(* PLC project factoryx.project, Bedrock IDE Bedrock IDE V1.4 *)
(* stored: creationDateTime 2017-02-21T09:02:52.9855728, modificationDateTime 2017-02-21T09:02:15.4674269 *)

TYPE EM_I_OUT_COM : STRUCT
  Request : INT;
  Command : INT;
  Pressure_SP : REAL;
  Owner : INT;
  Status : INT;
  CM_error : BOOL;
  CM_error_no : DINT;
  q_bACTVIE : BOOL;
  Level : REAL;
  Pressure : REAL;
END_STRUCT;
END_TYPE

FUNCTION somefunction : INT
  VAR_INPUT
    arg1 : INT;
    arg2 : INT;
  END_VAR

            
          
END_FUNCTION

FUNCTION write_to_DB_DW : BOOL
  VAR_INPUT
    DB_NO : INT;
    Location : INT;
    Value : INT;
  END_VAR

            
          
END_FUNCTION

FUNCTION_BLOCK Valve
  VAR_INPUT
    Command : BOOL;
    Feedback_Open : BOOL;
    Feedback_Close : BOOL;
  END_VAR
  VAR_OUTPUT
    Opened : BOOL;
    Closed : BOOL;
    Monitoring_Error : BOOL;
    Command_Open : BOOL;
  END_VAR

                    
                  
END_FUNCTION_BLOCK

FUNCTION_BLOCK Motor
  VAR_INPUT
    Command_On : BOOL;
    Command_Off : BOOL;
    Auto : BOOL;
    Manual : BOOL;
    Feedback_On : BOOL;
    Remote : BOOL;
    Error : BOOL;
    Enable : BOOL;
    Repair : BOOL;
  END_VAR
  VAR_OUTPUT
    Running : BOOL;
    Stopped : BOOL;
    Command_Run : BOOL;
    Error_Mon : BOOL;
    Error_VFD : BOOL;
    Error_Out : BOOL;
  END_VAR

                    
                  
END_FUNCTION_BLOCK

FUNCTION_BLOCK Motor_VFD
  VAR_INPUT
    Command_On : BOOL;
    Command_Off : BOOL;
    Auto : BOOL;
    Manual : BOOL;
    Feedback_On : BOOL;
    Remote : BOOL;
    Error : BOOL;
    Enable : BOOL;
    Repair : BOOL;
  END_VAR
  VAR_OUTPUT
    Running : BOOL;
    Stopped : BOOL;
    Command_Run : BOOL;
    Error_MS : BOOL;
    Error_Out : BOOL;
  END_VAR

                    
                  
END_FUNCTION_BLOCK

FUNCTION_BLOCK AI
  VAR_INPUT
    wVal : REAL;
  END_VAR
  VAR_OUTPUT
    QfVal : REAL;
    LIM_QbAH : BOOL;
    LIM_QbWH : BOOL;
    LIM_QbWL : BOOL;
    LIM_QbAL : BOOL;
    QERR : BOOL;
  END_VAR

                    
                  
END_FUNCTION_BLOCK

FUNCTION_BLOCK DI
  VAR_INPUT
    i_bInp : BOOL;
  END_VAR
  VAR_OUTPUT
    QON : BOOL;
  END_VAR

                    
                  
END_FUNCTION_BLOCK

FUNCTION_BLOCK PID
  VAR_INPUT
    i_bPCmdAUT : BOOL;
    i_bPCmdMAN : BOOL;
    Operator_Setpoint : REAL;
    Set_SP : BOOL;
    i_bPCmdPID : BOOL;
    i_bPCmdOPE : BOOL;
    Output_Value : REAL;
    Set_Output : REAL;
    wVal : REAL;
  END_VAR
  VAR_OUTPUT
    QfVal : REAL;
    QERR : BOOL;
    Q_wOP : REAL;
  END_VAR

                    
                  
END_FUNCTION_BLOCK

FUNCTION_BLOCK EM_I_OUT
  VAR_INPUT
    scantime : REAL := 200.0;
    sampletime : REAL;
    em_id : INT;
    Request : INT;
    Command : INT;
    Pressure_SP : REAL;
    Pump_RUN : BOOL;
    Pump_QERR : BOOL;  (* - General Error *)
    Pump_EERR : BOOL;  (* - External Error *)
    FS01_PV : BOOL;  (* Flow Switch - Digital Measurement *)
    PIC01_PV : REAL;  (* Pressure Controller *)
    PIC01_ERR : BOOL;  (* Pressure Controller *)
    LT01_PV : REAL;  (* Level Transmitter (m) *)
    LT01_AHH : BOOL;  (* Level Transmitter (m) *)
    LT01_AH : BOOL;  (* Level Transmitter (m) *)
    LT01_AL : BOOL;  (* Level Transmitter (m) *)
    LT01_ALL : BOOL;  (* Level Transmitter (m) *)
    LT01_ERR : BOOL;  (* Level Transmitter (m) *)
    XV_Bottom_OPN : BOOL;  (* Automatic Bottom Valve *)
    XV_Bottom_CLS : BOOL;  (* Automatic Bottom Valve *)
    XV_Bottom_MERR : BOOL;  (* Automatic Bottom Valve *)
    BV_Bottom_OPN : BOOL;  (* Manual Bottom Valve *)
    BV_Bottom_CLS : BOOL;  (* Manual Bottom Valve *)
    BV_Bottom_MERR : BOOL;  (* Manual Bottom Valve *)
    BV_Tran_M04_OPN : BOOL;  (* Trnasfer Valve to M04 *)
    BV_Tran_M04_CLS : BOOL;  (* Trnasfer Valve to M04 *)
    BV_Tran_M04_MERR : BOOL;  (* Trnasfer Valve to M04 *)
  END_VAR
  VAR_OUTPUT
    steptime_s : REAL;
    steptime_m : REAL;
    steptime_h : REAL;
    steptime_s : REAL;
    steptime_m : REAL;
    steptime_h : REAL;
    first_scan : BOOL;
    last_scan : BOOL;
    error_index_db : BOOL;
    Owner : INT;
    Status : INT;
    CM_error : BOOL;
    CM_error_no : DINT;
    q_bACTVIE : BOOL;
    Level : REAL;
    Pressure : REAL;
    Pump_ON : BOOL;  (* - Switch Motor ON *)
    Pump_AUT : BOOL;  (* - Swtich Motor to AUTO *)
    PIC01_EXT : BOOL;  (* Pressure Controller - Switch to External Mode *)
    PIC01_SP : REAL;  (* Pressure Controller - Operator Setpoint in Internal Mode *)
    PIC01_AUT : BOOL;  (* Pressure Controller - Switch to Auto Mode *)
    PIC01_VAL_OUT : REAL;  (* Pressure Controller - Operator Output Value *)
    PIC01_SET_SP : BOOL;  (* Pressure Controller *)
    PIC01_SET_OUT : BOOL;  (* Pressure Controller *)
    XV_Bottom_CMD : BOOL;  (* Automatic Bottom Valve - Auto command from program *)
    BV_Bottom_CMD : BOOL;  (* Manual Bottom Valve - Auto command from program *)
    BV_Tran_M04_CMD : BOOL;  (* Trnasfer Valve to M04 - Auto command from program *)
  END_VAR
  VAR
    first_scan : BOOL;
    last_scan : BOOL;
    previous_Command : INT;
    SP_PV : EM_I_OUT_COM;
  END_VAR
  VAR_TEMP
    initial_scan : BOOL;
  END_VAR

                    

					
// Copy all Setpoints from the COM
//--------------------------------
// 
//--------------------------------


Request:= SP_PV.Request;
Command:= SP_PV.Command;
Pressure_SP:= SP_PV.Pressure_SP;


// Acquiring logic
//--------------------------------
// 
//--------------------------------

Owner:= Request;


// Steptimers
//--------------------------------
// If the previous Command is not the same as the current one
// then reset the timers, else increase them
// This is at the start of the FB because normal commandchanges will take
// till the next cycle to become active
//--------------------------------

// if Command not changed then increase steptimer
IF (Command = previous_Command) THEN
	
	steptime_s:= steptime_s + scantime;

// else reset it at the start of a new step	
ELSE

	steptime_s:= 0.0;	
	
END_IF

// calculate the other two timers
steptime_m:= steptime_s / 60.0;
steptime_h:= steptime_m / 60.0;
		

		
// detect initial scan
//--------------------------------
// create a pulse active on the first cycle of a new scan
// this signal can be used in the step to execute some actions in the first cycle of the step
//--------------------------------

initial_scan:= Command <> previous_Command;		


// Save old step
//--------------------------------
// Save old step
//--------------------------------

previous_Command := Command;
		
		
// Collect the errors from the CMs
//--------------------------------
//
//--------------------------------
CM_Error:= (
	Pump_QERR
	OR Pump_EERR
	OR PIC01_ERR
	OR LT01_ERR
	OR XV_Bottom_MERR
	OR BV_Bottom_MERR
	OR BV_Tran_M04_MERR
);		
	

// Assign a message number to each error
//--------------------------------
// This code tries to assign an error message to each CM error
// If multiple CMs have an error then it only stores one
// This is the EM type so we don't know which CM/EM instance is connected
// So the error only contains the general name of the CM/EM instance
// If the actual name needs to be shown then it could be deducted
// at a higher level using the CM/EM name and EM instance 
//--------------------------------

// todo	


// START OF THE STATES
//################################
//################################
// Placeholder network to indicate the start of the actual sequence
//################################	  
//################################
// Step 0
//___EM_I_OUT_Step_0_
//================================
 
//================================	  

IF (Command = 0) THEN

	
	IF (first_scan) THEN
	
		// --- FIRST SCAN ---
		

	ELSE
	
		// --- CONTINUOUS ---
		

		// Action: stop Pump
		Pump_ON:= false;

		// Action: close XV_Bottom
		XV_Bottom_CMD:= false;

		// Action: close BV_Bottom
		BV_Bottom_CMD:= false;

		// Action: close BV_Tran_M04
		BV_Tran_M04_CMD:= false;

	END_IF
	

	// --- CONDITIONS ---
	IF (
		XV_Bottom_CLS
		AND BV_Bottom_CLS
		AND BV_Tran_M04_CLS
	) THEN
	
		Status:= Command;
		
	END_IF
	
END_IF	

IF (previous_Command = 0 and Command <> 0 ) THEN		
	
	
	// --- LAST SCAN ---
	


END_IF 

	
// Step 1
//___EM_I_OUT_Step_1_
//================================
 
//================================	  

IF (Command = 1) THEN

	
	IF (first_scan) THEN
	
		// --- FIRST SCAN ---
		

	ELSE
	
		// --- CONTINUOUS ---
		

		// Action: stop Pump
		Pump_ON:= false;

		// Action: open XV_Bottom
		XV_Bottom_CMD:= true;

	END_IF
	

	// --- CONDITIONS ---
	IF (
		XV_Bottom_OPN
	) THEN
	
		Status:= Command;
		
	END_IF
	
END_IF	

IF (previous_Command = 1 and Command <> 1 ) THEN		
	
	
	// --- LAST SCAN ---
	


END_IF 

	
// Step 2
//___EM_I_OUT_Step_2_
//================================
 
//================================	  

IF (Command = 2) THEN

	
	IF (first_scan) THEN
	
		// --- FIRST SCAN ---
		

		// Action: PIC01_SP = 10.0
		PIC01_SP:= 10.0;

		// Action: PIC01_SET_SP = true
		PIC01_SET_SP:= true;

	ELSE
	
		// --- CONTINUOUS ---
		

		// Action: start Pump
		Pump_ON:= true;

		// Action: auto 10.0 bar PIC01
		PIC01_AUT:= true;

		// Action: open XV_Bottom
		XV_Bottom_CMD:= true;

		// Action: PIC01_SET_SP = false
		PIC01_SET_SP:= false;

	END_IF
	

	// --- CONDITIONS ---
	IF (
		Pump_RUN
		AND XV_Bottom_OPN
	) THEN
	
		Status:= Command;
		
	END_IF
	
END_IF	

IF (previous_Command = 2 and Command <> 2 ) THEN		
	
	
	// --- LAST SCAN ---
	


END_IF 

	
// Step 3
//___EM_I_OUT_Step_3_
//================================
 
//================================	  

IF (Command = 3) THEN

	
	IF (first_scan) THEN
	
		// --- FIRST SCAN ---
		

	ELSE
	
		// --- CONTINUOUS ---
		

		// Action: stop Pump
		Pump_ON:= false;

		// Action: open BV_Bottom
		BV_Bottom_CMD:= true;

		// Action: open BV_Tran_M04
		BV_Tran_M04_CMD:= true;

	END_IF
	

	// --- CONDITIONS ---
	IF (
		BV_Bottom_OPN
		AND BV_Tran_M04_OPN
	) THEN
	
		Status:= Command;
		
	END_IF
	
END_IF	

IF (previous_Command = 3 and Command <> 3 ) THEN		
	
	
	// --- LAST SCAN ---
	


END_IF 

	
// Step 4
//___EM_I_OUT_Step_4_
//================================
 
//================================	  

IF (Command = 4) THEN

	
	IF (first_scan) THEN
	
		// --- FIRST SCAN ---
		

		// Action: PIC01_SP = Pressure_SP
		PIC01_SP:= Pressure_SP;

		// Action: PIC01_SET_SP = true
		PIC01_SET_SP:= true;

	ELSE
	
		// --- CONTINUOUS ---
		

		// Action: start Pump
		Pump_ON:= true;

		// Action: auto Pressure_SP PIC01
		PIC01_AUT:= true;

		// Action: open BV_Bottom
		BV_Bottom_CMD:= true;

		// Action: open BV_Tran_M04
		BV_Tran_M04_CMD:= true;

		// Action: PIC01_SET_SP = false
		PIC01_SET_SP:= false;

	END_IF
	

	// --- CONDITIONS ---
	IF (
		Pump_RUN
		AND BV_Bottom_OPN
		AND BV_Tran_M04_OPN
	) THEN
	
		Status:= Command;
		
	END_IF
	
END_IF	

IF (previous_Command = 4 and Command <> 4 ) THEN		
	
	
	// --- LAST SCAN ---
	


END_IF 

	
// Step 5
//___EM_I_OUT_Step_5_
//================================
 
//================================	  

IF (Command = 5) THEN

	
	IF (first_scan) THEN
	
		// --- FIRST SCAN ---
		

		// Action: PIC01_VAL_OUT = 20.0
		PIC01_VAL_OUT:= 20.0;

		// Action: PIC01_SET_OUT = true
		PIC01_SET_OUT:= true;

	ELSE
	
		// --- CONTINUOUS ---
		

		// Action: start Pump
		Pump_ON:= true;

		// Action: manual 20.0 Hz PIC01
		PIC01_AUT:= false;

		// Action: open XV_Bottom
		XV_Bottom_CMD:= true;

		// Action: PIC01_SET_OUT = false
		PIC01_SET_OUT:= false;

	END_IF
	

	// --- CONDITIONS ---
	IF (
		Pump_RUN
		AND XV_Bottom_OPN
	) THEN
	
		Status:= Command;
		
	END_IF
	
END_IF	

IF (previous_Command = 5 and Command <> 5 ) THEN		
	
	
	// --- LAST SCAN ---
	


END_IF 

	




// END OF THE STATES
//################################
//################################
// Placeholder network to indicate the end of the actual sequence
//################################	  
//################################


// General Actions - After
//--------------------------------
// General Actions - After
//--------------------------------

		// Action: Level = LT01
		Level:= LT01_PV;

		// Action: Pressure = PIC01
		Pressure:= PIC01_PV;
// Copy all Process Values to the UDT
//--------------------------------
// 
//--------------------------------


SP_PV.Owner:= Owner;
SP_PV.Status:= Status;
SP_PV.CM_error:= CM_error;
SP_PV.CM_error_no:= CM_error_no;
SP_PV.q_bACTVIE:= q_bACTVIE;
SP_PV.Level:= Level;
SP_PV.Pressure:= Pressure;


// Clean up request
//--------------------------------
// Phases don't clean up their requests on the EM side
// So at the end of the EM reset the request
// If the phase is still there then it will write the request again by the next scan
//--------------------------------
	
request:= 0;

					
                  
END_FUNCTION_BLOCK

FUNCTION_BLOCK phase_example
  VAR_INPUT
    scantime : REAL := 200.0;
    scantime : REAL;
    Bool1 : BOOL;
    Bool2 : BOOL;
    DB_NO : INT;
    XV003_OPN : BOOL;
    XV003_CLS : BOOL;
    XV003_MERR : BOOL;
    XV004_OPN : BOOL;
    XV004_CLS : BOOL;
    XV004_MERR : BOOL;
    XV005_OPN : BOOL;
    XV005_CLS : BOOL;
    XV005_MERR : BOOL;
    P001_RUN : BOOL;  (* test a CM *)
    P001_STOP : BOOL;  (* test a CM *)
    P001_MERR : BOOL;  (* test a CM *)
    P001_MPS : BOOL;  (* test a CM - Motor Protecting Switch *)
    P002_RUN : BOOL;  (* test a CM where the casing doesn't match an existing type *)
    P002_STOP : BOOL;  (* test a CM where the casing doesn't match an existing type *)
    P002_MERR : BOOL;  (* test a CM where the casing doesn't match an existing type *)
    P002_MPS : BOOL;  (* test a CM where the casing doesn't match an existing type - Motor Protecting Switch *)
    EM_I_OUT_ID : INT;  (* fixed value linked to input *)
    LT001_PV : REAL;
    LT001_AHH : BOOL;
    LT001_AH : BOOL;
    LT001_AL : BOOL;
    LT001_ALL : BOOL;
    LT001_ERR : BOOL;
    LT002_PV : REAL;
    LT002_AHH : BOOL;
    LT002_AH : BOOL;
    LT002_AL : BOOL;
    LT002_ALL : BOOL;
    LT002_ERR : BOOL;
    FIC001_PV : REAL;
    FIC001_ERR : BOOL;
    Some_Dyn_EM_AUT : INT;  (* EM ID: selection based on route or recipy *)
    XV008_OPN : BOOL;
    XV008_CLS : BOOL;
    XV008_MERR : BOOL;
  END_VAR
  VAR_OUTPUT
    phase_id : INT;
    state : INT;
    stepnumber : INT;
    message : DINT;
    button_1_text : DINT;
    button_2_text : DINT;
    button_3_text : DINT;
    button_1_visible : BOOL;
    button_2_visible : BOOL;
    button_3_visible : BOOL;
    state_idle : BOOL;
    state_running : BOOL;
    state_complete : BOOL;
    state_pausing : BOOL;
    state_paused : BOOL;
    state_holding : BOOL;
    state_held : BOOL;
    state_restarting : BOOL;
    state_stopping : BOOL;
    state_stopped : BOOL;
    state_aborting : BOOL;
    state_aborted : BOOL;
    enable_start : BOOL;
    enable_stop : BOOL;
    enable_hold : BOOL;
    enable_restart : BOOL;
    enable_abort : BOOL;
    enable_reset : BOOL;
    enable_pause : BOOL;
    enable_resume : BOOL;
    enable_auto : BOOL;
    enable_man : BOOL;
    enable_byte : BYTE;
    auto : BOOL;
    steptime_s : REAL;
    steptime_m : REAL;
    steptime_h : REAL;
    message_number_01 : DINT;
    message_number_02 : DINT;
    message_number_03 : DINT;
    message_number_04 : DINT;
    message_number_05 : DINT;
    message_number_06 : DINT;
    message_number_07 : DINT;
    message_number_08 : DINT;
    message_number_09 : DINT;
    message_number_10 : DINT;
    phase_id : INT;
    state : INT;
    stepnumber : INT;
    message : DINT;
    button_1_text : DINT;
    button_2_text : DINT;
    button_3_text : DINT;
    button_1_visible : BOOL;
    button_2_visible : BOOL;
    button_3_visible : BOOL;
    state_idle : BOOL;
    state_running : BOOL;
    state_complete : BOOL;
    state_pausing : BOOL;
    state_paused : BOOL;
    state_holding : BOOL;
    state_held : BOOL;
    state_restarting : BOOL;
    state_stopping : BOOL;
    state_stopped : BOOL;
    state_aborting : BOOL;
    state_aborted : BOOL;
    enable_start : INT;
    enable_stop : INT;
    enable_hold : INT;
    enable_restart : INT;
    enable_abort : INT;
    enable_reset : INT;
    enable_pause : INT;
    enable_resume : INT;
    enable_auto : BOOL;
    enable_man : BOOL;
    auto : BOOL;
    steptime_s : REAL;
    steptime_m : REAL;
    steptime_h : REAL;
    MSG_no01 : DINT;
    MSG_no02 : DINT;
    MSG_no03 : DINT;
    MSG_no04 : DINT;
    MSG_no05 : DINT;
    MSG_no06 : DINT;
    MSG_no07 : DINT;
    MSG_no08 : DINT;
    MSG_no09 : DINT;
    MSG_no10 : DINT;
    Destination : INT;
    setpoint : REAL;
    some_bool_out : BOOL;
    XV003_CMD : BOOL;  (* - Auto command from program *)
    XV004_CMD : BOOL;  (* - Auto command from program *)
    XV005_CMD : BOOL;  (* - Auto command from program *)
    P001_ON : BOOL;  (* test a CM - Switch Motor ON *)
    P001_AUT : BOOL;  (* test a CM - Swtich Motor to AUTO *)
    P002_ON : BOOL;  (* test a CM where the casing doesn't match an existing type - Switch Motor ON *)
    P002_AUT : BOOL;  (* test a CM where the casing doesn't match an existing type - Swtich Motor to AUTO *)
    FIC001_EXT : BOOL;  (* - Switch to External Mode *)
    FIC001_SP : REAL;  (* - Operator Setpoint in Internal Mode *)
    FIC001_AUT : BOOL;  (* - Switch to Auto Mode *)
    FIC001_VAL_OUT : REAL;  (* - Operator Output Value *)
    FIC001_SET_SP : BOOL;
    FIC001_SET_OUT : BOOL;
    Some_Dyn_EM_ID : INT;  (* EM ID: receives value from _AUT or _MN, depending on the mode of the sequence *)
    timer_dosing_pause : BOOL;  (* timer paused *)
    timer_dosing_s : REAL;  (* timer in seconds *)
    timer_dosing_m : REAL;  (* timer in minutes *)
    timer_dosing_h : REAL;  (* timer in hours *)
    timer_mixing_pause : BOOL;  (* timer paused *)
    timer_mixing_s : REAL;  (* timer in seconds *)
    timer_mixing_m : REAL;  (* timer in minutes *)
    timer_mixing_h : REAL;  (* timer in hours *)
    timer_circulation_pause : BOOL;  (* timer paused *)
    timer_circulation_s : REAL;  (* timer in seconds *)
    timer_circulation_m : REAL;  (* timer in minutes *)
    timer_circulation_h : REAL;  (* timer in hours *)
    XV008_CMD : BOOL;  (* - Auto command from program *)
  END_VAR
  VAR
    hmi_commands : INT;
    previous_stepnumber : INT;
    start_conditions : BOOL;
    hold_conditions : BOOL;
    first_scan : BOOL;
    last_scan : BOOL;
    start_cond_01 : BOOL;
    start_cond_02 : BOOL;
    start_cond_03 : BOOL;
    start_cond_04 : BOOL;
    start_cond_05 : BOOL;
    start_cond_06 : BOOL;
    start_cond_07 : BOOL;
    start_cond_08 : BOOL;
    start_cond_09 : BOOL;
    start_cond_10 : BOOL;
    start_cond_11 : BOOL;
    start_cond_12 : BOOL;
    start_cond_13 : BOOL;
    start_cond_14 : BOOL;
    start_cond_15 : BOOL;
    start_cond_16 : BOOL;
    hold_cond_01 : BOOL;
    hold_cond_02 : BOOL;
    hold_cond_03 : BOOL;
    hold_cond_04 : BOOL;
    hold_cond_05 : BOOL;
    hold_cond_06 : BOOL;
    hold_cond_07 : BOOL;
    hold_cond_08 : BOOL;
    hold_cond_09 : BOOL;
    hold_cond_10 : BOOL;
    hold_cond_11 : BOOL;
    hold_cond_12 : BOOL;
    hold_cond_13 : BOOL;
    hold_cond_14 : BOOL;
    hold_cond_15 : BOOL;
    hold_cond_16 : BOOL;
    in_steprange : BOOL;
    Module_Error : BOOL;
    CM_Error_no : BOOL;
    EM_Error_no : BOOL;
    plc_commands : DWORD;
    hmi_commands : DWORD;
    Some_Dyn_EM_MN : INT;  (* EM ID: direct EM selection from HMI *)
    hmi_par_without_unit : REAL;
    timesetting : REAL;
    previous_stepnumber : INT;
    start_conditions : BOOL;
    hold_conditions : BOOL;
    first_scan : BOOL;
    last_scan : BOOL;
    start_cond_01 : BOOL;
    start_cond_02 : BOOL;
    start_cond_03 : BOOL;
    start_cond_04 : BOOL;
    start_cond_05 : BOOL;
    start_cond_06 : BOOL;
    start_cond_07 : BOOL;
    start_cond_08 : BOOL;
    start_cond_09 : BOOL;
    start_cond_10 : BOOL;
    start_cond_11 : BOOL;
    start_cond_12 : BOOL;
    start_cond_13 : BOOL;
    start_cond_14 : BOOL;
    start_cond_15 : BOOL;
    start_cond_16 : BOOL;
    hold_cond_01 : BOOL;
    hold_cond_02 : BOOL;
    hold_cond_03 : BOOL;
    hold_cond_04 : BOOL;
    hold_cond_05 : BOOL;
    hold_cond_06 : BOOL;
    hold_cond_07 : BOOL;
    hold_cond_08 : BOOL;
    hold_cond_09 : BOOL;
    hold_cond_10 : BOOL;
    hold_cond_11 : BOOL;
    hold_cond_12 : BOOL;
    hold_cond_13 : BOOL;
    hold_cond_14 : BOOL;
    hold_cond_15 : BOOL;
    hold_cond_16 : BOOL;
    in_steprange : BOOL;
    Module_Error : BOOL;
    CM_Error_no : DINT;
    EM_Error_no : DINT;
    plc_start : BOOL;
    plc_stop : BOOL;
    plc_hold : BOOL;
    plc_restart : BOOL;
    plc_abort : BOOL;
    plc_reset : BOOL;
    plc_pause : BOOL;
    plc_resume : BOOL;
    plc_auto : BOOL;
    plc_man : BOOL;
    hmi_start : INT;
    hmi_stop : INT;
    hmi_hold : INT;
    hmi_restart : INT;
    hmi_abort : INT;
    hmi_reset : INT;
    hmi_pause : INT;
    hmi_resume : INT;
    hmi_auto : BOOL;
    hmi_man : BOOL;
    hmi_BTN1 : BOOL;
    hmi_BTN2 : BOOL;
    hmi_BTN3 : BOOL;
    command_start : BOOL;
    command_stop : BOOL;
    command_hold : BOOL;
    command_restart : BOOL;
    command_abort : BOOL;
    command_reset : BOOL;
    command_pause : BOOL;
    command_resume : BOOL;
    command_auto : BOOL;
    command_man : BOOL;
    button_1_pushed : BOOL;
    button_2_pushed : BOOL;
    button_3_pushed : BOOL;
    sh_cond_01 : INT;
    sh_cond_02 : INT;
    sh_cond_03 : INT;
    sh_cond_04 : INT;
    sh_cond_05 : INT;
    sh_cond_06 : INT;
    sh_cond_07 : INT;
    sh_cond_08 : INT;
    sh_cond_09 : INT;
    sh_cond_10 : INT;
    sh_cond_11 : INT;
    sh_cond_12 : INT;
    sh_cond_13 : INT;
    sh_cond_14 : INT;
    sh_cond_15 : INT;
    sh_cond_16 : INT;
    initial_scan : BOOL;
    Temp_stepnumber : INT;
    e : REAL;
    f : REAL;
    g : REAL;
    h : REAL;
    ii : REAL;
    j : REAL;
    k : REAL;
    l : REAL;
    mm : REAL;
    n : REAL;
    o : REAL;
    pp : REAL;
    qq : REAL;
    rr : REAL;
    ss : REAL;
    tt : REAL;
    u : REAL;
    v : REAL;
    ww : REAL;
    xx : REAL;
    y : REAL;
    z : REAL;
    foo : REAL;
    bar : REAL;
    stoplevel : REAL;
    startlevel : REAL;
    offset : REAL;
    var1 : REAL;
    test1 : REAL;
    test2 : REAL;
    intvar : INT;
    EM_I_OUT : EM_I_OUT_COM;  (* Structure linking the EM *)
    EM_I_OUT_POINTER : POINTER TO EM_I_OUT_COM;  (* Pointer needed for dereferencing the linked STRUCT *)
    Some_Dyn_EM : EM_I_OUT_COM;  (* Structure linking the EM *)
    Some_Dyn_EM_POINTER : POINTER TO EM_I_OUT_COM;  (* Pointer needed for dereferencing the linked STRUCT *)
  END_VAR
  VAR_TEMP
    plc_start : BOOL;
    plc_stop : BOOL;
    plc_hold : BOOL;
    plc_restart : BOOL;
    plc_abort : BOOL;
    plc_reset : BOOL;
    plc_pause : BOOL;
    plc_resume : BOOL;
    plc_auto : BOOL;
    plc_man : BOOL;
    plc_cmd : BOOL;
    hmi_start : BOOL;
    hmi_stop : BOOL;
    hmi_hold : BOOL;
    hmi_restart : BOOL;
    hmi_abort : BOOL;
    hmi_reset : BOOL;
    hmi_pause : BOOL;
    hmi_resume : BOOL;
    hmi_auto : BOOL;
    hmi_man : BOOL;
    hmi_cmd : BYTE;
    command_start : BOOL;
    command_stop : BOOL;
    command_hold : BOOL;
    command_restart : BOOL;
    command_abort : BOOL;
    command_reset : BOOL;
    command_pause : BOOL;
    command_resume : BOOL;
    command_auto : BOOL;
    command_man : BOOL;
    command_byte : BYTE;
    button_1_pushed : BOOL;
    button_2_pushed : BOOL;
    button_3_pushed : BOOL;
    sh_cond_01 : BOOL;
    sh_cond_02 : BOOL;
    sh_cond_03 : BOOL;
    sh_cond_04 : BOOL;
    sh_cond_05 : BOOL;
    sh_cond_06 : BOOL;
    sh_cond_07 : BOOL;
    sh_cond_08 : BOOL;
    sh_cond_09 : BOOL;
    sh_cond_10 : BOOL;
    sh_cond_11 : BOOL;
    sh_cond_12 : BOOL;
    sh_cond_13 : BOOL;
    sh_cond_14 : BOOL;
    sh_cond_15 : BOOL;
    sh_cond_16 : BOOL;
    initial_scan : BOOL;
    current_stepnumber : INT;
  END_VAR

                    

// INDEX
//--------------------------------
//___phase_example_Step_0_
//___phase_example_Step_10_
//___phase_example_Step_20_
//___phase_example_Step_30_
//___phase_example_Step_40_
//___phase_example_Step_50_
//___phase_example_Step_70_
//___phase_example_Step_80_
//___phase_example_Step_90_
//___phase_example_Step_100_
//___phase_example_Step_120_
//___phase_example_Step_130_
//___phase_example_Step_150_
//___phase_example_Step_170_
//___phase_example_Step_180_
//___phase_example_Step_190_
//___phase_example_Step_200_
//___phase_example_Step_230_
//___phase_example_Step_250_
//___phase_example_Step_260_
//___phase_example_Step_280_
//___phase_example_Step_300_
//___phase_example_Step_310_
//___phase_example_Step_320_
//___phase_example_Step_330_
//___phase_example_Step_340_
//___phase_example_Step_350_
//___phase_example_Step_360_
//___phase_example_Step_370_
//___phase_example_Step_420_
//___phase_example_Step_430_
//___phase_example_Step_440_
//___phase_example_Step_450_
//___phase_example_Step_460_
//___phase_example_Step_470_
//___phase_example_Step_480_
//___phase_example_Step_490_
//___phase_example_Step_510_
//___phase_example_Step_520_
//___phase_example_Step_530_
//___phase_example_Step_540_
//___phase_example_Step_550_
//___phase_example_Step_560_
//___phase_example_Step_570_
//___phase_example_Step_580_
//___phase_example_Step_590_
//___phase_example_Step_600_
//___phase_example_Step_610_
//___phase_example_Step_640_
//___phase_example_Step_650_
//___phase_example_Step_660_
//___phase_example_Step_670_
//___phase_example_Step_680_
//___phase_example_Step_690_
//___phase_example_Step_700_
//___phase_example_Step_710_
//___phase_example_Step_720_
//___phase_example_Step_730_
//___phase_example_Step_740_
//___phase_example_Step_750_
//___phase_example_Step_760_
//___phase_example_Step_770_
//___phase_example_Step_780_
//___phase_example_Step_790_
//___phase_example_Step_810_
//___phase_example_Step_820_
//___phase_example_Step_830_
//___phase_example_Step_840_
//___phase_example_Step_850_
//___phase_example_Step_860_
//___phase_example_Step_870_
//___phase_example_Step_880_
//___phase_example_Step_890_
//___phase_example_Step_910_
//___phase_example_Step_920_
//___phase_example_Step_930_
//___phase_example_Step_940_
//___phase_example_Step_950_
//___phase_example_Step_960_
//___phase_example_Step_970_
//___phase_example_Step_980_
//___phase_example_Step_990_
//___phase_example_Step_1000_
//___phase_example_Step_8000_
//--------------------------------				
		
		
// Read EMs
//--------------------------------
//
//--------------------------------

// todo: protect againt not a pointer
	   
EM_I_OUT_Pointer:=cstate.EM_Index[EM_I_OUT_ID];
EM_I_OUT := EM_I_OUT_Pointer^;
	   
Some_Dyn_EM_Pointer:=cstate.EM_Index[Some_Dyn_EM_ID];
Some_Dyn_EM := Some_Dyn_EM_Pointer^;



// HMI Commands
//--------------------------------
// Get the commands from the HMI that have been received in the last cycle
// They come in a DWORD to save tags
// They need to be transferred to BOOLS for easy use
// Once transferred then clear the DWORD so new commands can be detected in the next cycle
//--------------------------------
hmi_start:= hmi_commands.0;
hmi_stop:= hmi_commands.1;
hmi_restart:= hmi_commands.2;
hmi_abort:= hmi_commands.3;
hmi_reset:= hmi_commands.4;
hmi_pause:= hmi_commands.5;
hmi_resume:= hmi_commands.6;
hmi_auto:= hmi_commands.7;
hmi_man:= hmi_commands.8;
button_1_pushed:= hmi_commands.9;
button_2_pushed:= hmi_commands.10;
button_3_pushed:= hmi_commands.11;

// clear the command
hmi_commands:= 0;


// Combined Commands
//--------------------------------
// Combine the commands from the HMI and PLC in one command
// (OR-function)
//--------------------------------

command_start := hmi_start OR plc_start;
command_stop := hmi_stop OR plc_stop;
command_hold := hmi_hold OR plc_hold;
command_restart := hmi_restart OR plc_restart;
command_abort := hmi_abort OR plc_abort;
command_reset := hmi_reset OR plc_reset;
command_pause := hmi_pause OR plc_pause;
command_resume := hmi_resume OR plc_resume;
command_auto := hmi_auto OR plc_auto;
command_man := hmi_man OR plc_man;

IF (command_auto) THEN
	auto:= TRUE;
END_IF

IF (command_man) THEN
	auto:= FALSE;
END_IF

IF (auto) THEN
	enable_man:= TRUE;
	enable_auto:= FALSE;
ELSE
	enable_man:= FALSE;
	enable_auto:= TRUE;
END_IF



// Steptimers
//--------------------------------
// If the previous stepnumber is not the same as the current one
// then reset the timers, else increase them
// This is at the start of the FB because normal stepchanges will take
// till the next cycle to become active
//--------------------------------

// if stepnumber not changed then increase it
IF (stepnumber = previous_stepnumber) THEN
	
	steptime_s:= steptime_s + scantime;

// else reset it at the start of a new step	
ELSE

	steptime_s:= 0.0;	
	
END_IF

// calculate the other two timers
steptime_m:= steptime_s / 60.0;
steptime_h:= steptime_m / 60.0;


// Other Timers
//--------------------------------
// If timers are needed that cannot be solved with the steptime.
// Timers need to start with the name 'timer'
// They are paused by default
// They can be unpaused
// They can be reset by writing the value to 0 in the action
// Every timer is available in s, m and h
//--------------------------------

//--------------------------------
// timer_dosing
//--------------------------------

// if not paused...
IF (NOT timer_dosing_pause) THEN

	timer_dosing_s:= timer_dosing_s + scantime;

END_IF

// calculate the other two timers
timer_dosing_m:= timer_dosing_s / 60.0;
timer_dosing_h:= timer_dosing_m / 60.0;

//--------------------------------
// timer_mixing
//--------------------------------

// if not paused...
IF (NOT timer_mixing_pause) THEN

	timer_mixing_s:= timer_mixing_s + scantime;

END_IF

// calculate the other two timers
timer_mixing_m:= timer_mixing_s / 60.0;
timer_mixing_h:= timer_mixing_m / 60.0;

//--------------------------------
// timer_circulation
//--------------------------------

// if not paused...
IF (NOT timer_circulation_pause) THEN

	timer_circulation_s:= timer_circulation_s + scantime;

END_IF

// calculate the other two timers
timer_circulation_m:= timer_circulation_s / 60.0;
timer_circulation_h:= timer_circulation_m / 60.0;



// detect initial scan
//--------------------------------
// create a pulse active on the first cycle of a new scan
// this signal can be used in the step to execute some actions in the first cycle of the step
//--------------------------------

initial_scan:= stepnumber <> previous_stepnumber;


// Save old step
//--------------------------------
// Save old step
//--------------------------------

previous_stepnumber := stepnumber;

// Save current step
//--------------------------------
// This is used to detect a stepnumber change in the step
// for example used to execute the last scan
//--------------------------------

current_stepnumber := stepnumber;


// Change States
//--------------------------------
// Change States
//--------------------------------
// This phase template is design to let the stepnumber be the single
// source of truth for the state of the phase.
// All other indicators of state from this phase are deducted from the
// stepnumber.
// And the state can only be changed by changing the stepnumber 
//
// For every state we both create a bit, and an integer value
// Both have the same meaning and can be chosen for usage based
// on what is most convenient
//--------------------------------


// Stop Command
IF (enable_stop AND command_stop) THEN
	
	stepnumber:= 0;

END_IF

// Hold Command
IF (enable_hold AND (command_hold OR NOT hold_conditions)) THEN
	
	stepnumber:= 8000;

END_IF

// Abort Command
IF (enable_abort AND command_abort) THEN
	
	stepnumber:= 9000;

END_IF

// Pause Command
IF (enable_pause AND command_pause) THEN
	
	stepnumber:= 6000;

END_IF


// Phase States
//--------------------------------
// Update Phase States based on the stepnumber
// 0 idle 
// 1 running
// 2 completed
// 3 pausing
// 4 paused
// 5 holding
// 6 held
// 7 restarting
// 8 stopping
// 9 stopped
// 10 aborting
// 11 aborted
//--------------------------------
// See above for explanation
//--------------------------------


//--------------------------------
// Disable all permissions for the commands
// The individial permissions will be set again
// in the next steps depending on the state
//--------------------------------

enable_start:= FALSE;
enable_stop:= FALSE;
enable_hold:= FALSE;
enable_restart:= FALSE;
// enable_abort:= FALSE;
enable_reset:= FALSE;
enable_pause:= FALSE;
enable_resume:= FALSE;


// 0 Idle state based on stepnumber
IF (stepnumber >= 0 AND stepnumber <= 0) THEN
	
	state_idle:= TRUE;
	state:= 0;
	enable_start:= TRUE;

END_IF

// 1 Running state based on stepnumber
IF (stepnumber >= 1 AND stepnumber <= 9999) THEN
	
	state_running := TRUE;
	state:= 1;
	enable_stop:= TRUE;
	enable_hold:= TRUE;
// enable_abort:= TRUE;
	enable_pause:= TRUE;

END_IF

// 2 Completed state based on stepnumber
IF (stepnumber >= 700 AND stepnumber <= 1000) THEN
	
	state_complete:= TRUE;
	state:= 2;
	enable_reset:= TRUE;

END_IF

// 3 Pausing state based on stepnumber
IF (stepnumber >= 6000 AND stepnumber <= 6900) THEN
	
	state_pausing:= TRUE;
	state:= 3;
	enable_stop:= TRUE;
	enable_hold:= TRUE;
// enable_abort:= TRUE;	
	
END_IF

// 4 Paused state based on stepnumber
IF (stepnumber >= 6900 AND stepnumber <= 6999) THEN
	
	state_paused:= TRUE;
	state:= 4;
	enable_stop:= TRUE;
	enable_hold:= TRUE;
// enable_abort:= TRUE;	
	enable_resume:= TRUE;
	
END_IF

// 5 Holding state based on stepnumber
IF (stepnumber >= 8000 AND stepnumber <= 8900) THEN
	
	state_holding:= TRUE;
	state:= 5;
	enable_stop:= TRUE;
// enable_abort:= TRUE;	
	
END_IF

// 6 Held state based on stepnumber
IF (stepnumber >= 8900 AND stepnumber <= 8999) THEN
	
	state_held:= TRUE;
	state:= 6;
	enable_stop:= TRUE;
	enable_restart:= TRUE;
	enable_abort:= TRUE;
	
END_IF

// 7 Restarting state based on stepnumber
IF (stepnumber >= 5000 AND stepnumber <= 5900) THEN
	
	state_restarting:= TRUE;
	state:= 7;
	enable_stop:= TRUE;
	enable_hold:= TRUE;
// enable_abort:= TRUE;
	
END_IF

// 8 Stopping state based on stepnumber
IF (stepnumber >= 7000 AND stepnumber <= 7900) THEN
	
	state_stopping:= TRUE;
	state:= 8;
// enable_abort:= TRUE;
	
END_IF

// 9 Stopped state based on stepnumber
IF (stepnumber >= 7900 AND stepnumber <= 7999) THEN
	
	state_stopped:= TRUE;
	state:= 9;
// enable_abort:= TRUE;
	enable_reset:= TRUE;
	
END_IF

// 10 Aborting state based on stepnumber
IF (stepnumber >= 9000 AND stepnumber <= 9900) THEN
	
	state_aborting:= TRUE;
	state:= 10;

END_IF

// 11 Aborted state based on stepnumber
IF(stepnumber >= 9900 AND stepnumber <= 9999) THEN
	
	state_aborted:= TRUE;
	state:= 11;
	enable_reset:= TRUE;

END_IF


// Disable start command if start_conditions are not ok
IF (NOT start_conditions) THEN
	
	enable_start:= FALSE;

END_IF


// Collect the errors from the connected Modules (CMs and EMs)
//--------------------------------
//
//--------------------------------
Module_Error:= (
	XV003_MERR
	OR XV004_MERR
	OR XV005_MERR
	OR P001_MERR
	OR P001_MPS
	OR P002_MERR
	OR P002_MPS
	OR LT001_ERR
	OR LT002_ERR
	OR FIC001_ERR
	OR XV008_MERR
);

// Assign a message number to each error
//--------------------------------
// This code tries to assign an error message to each CM error
// If multiple CMs have an error then it only stores one
// This is the phase type so we don't know which CM/EM instance is connected
// So the error only contains the general name of the CM/EM instance
// If the actual name needs to be shown then it could be deducted
// at a higher level using the CM/EM name and phase instance 
//--------------------------------

// todo

// Start and Hold Conditions
//--------------------------------
// 
//--------------------------------

start_conditions:= FALSE;
hold_conditions:= FALSE; // TRUE = safe condition


// START OF THE STEPS AND TRANSITIONS
//################################
//################################
// Placeholder network to indicate the start of the actual sequence
//################################	  
//################################



// Step 0
//___phase_example_Step_0_
//================================
// Test step with only a comment and transition 
//================================	  

IF (stepnumber = 0) THEN

	
	IF (first_scan) THEN
	
		// --- FIRST SCAN ---
		

	ELSE
	
		// --- CONTINUOUS ---
		

	END_IF
	
	
	// --- TRANSITION TO S10 ---
	IF (
		TRUE
	) THEN
	
		stepnumber:= 10;
		
	END_IF
		
		
		
	IF (stepnumber <> current_stepnumber) THEN
	
		// --- LAST SCAN ---
	
	
	END_IF
	

END_IF 

	


// Step 10
//___phase_example_Step_10_
//================================
// Test multiple comments
// this is another line 
//================================	  

IF (stepnumber = 10) THEN

	
	IF (first_scan) THEN
	
		// --- FIRST SCAN ---
		

	ELSE
	
		// --- CONTINUOUS ---
		

	END_IF
	
	
	// --- TRANSITION TO S20 ---
	IF (
		TRUE
	) THEN
	
		stepnumber:= 20;
		
	END_IF
		
		
		
	IF (stepnumber <> current_stepnumber) THEN
	
		// --- LAST SCAN ---
	
	
	END_IF
	

END_IF 

	
// Step 20
//___phase_example_Step_20_
//================================
// Test some spacing before the comment
// Test some spacing before the first comment word 
//================================	  

IF (stepnumber = 20) THEN

	
	IF (first_scan) THEN
	
		// --- FIRST SCAN ---
		

	ELSE
	
		// --- CONTINUOUS ---
		

	END_IF
	
	
	// --- TRANSITION TO S30 ---
	IF (
		TRUE
	) THEN
	
		stepnumber:= 30;
		
	END_IF
		
		
		
	IF (stepnumber <> current_stepnumber) THEN
	
		// --- LAST SCAN ---
	
	
	END_IF
	

END_IF 

	
// Step 30
//___phase_example_Step_30_
//================================
// test a simple assignment with a variable 
//================================	  

IF (stepnumber = 30) THEN

	
	IF (first_scan) THEN
	
		// --- FIRST SCAN ---
		

	ELSE
	
		// --- CONTINUOUS ---
		

		// Action: e = f
		e:= f;

	END_IF
	
	
	// --- TRANSITION TO S40 ---
	IF (
		TRUE
	) THEN
	
		stepnumber:= 40;
		
	END_IF
		
		
		
	IF (stepnumber <> current_stepnumber) THEN
	
		// --- LAST SCAN ---
	
	
	END_IF
	

END_IF 

	
// Step 40
//___phase_example_Step_40_
//================================
// test a simple assignment with a REAL 
//================================	  

IF (stepnumber = 40) THEN

	
	IF (first_scan) THEN
	
		// --- FIRST SCAN ---
		

	ELSE
	
		// --- CONTINUOUS ---
		

		// Action: setpoint = 25.0
		setpoint:= 25.0;

	END_IF
	
	
	// --- TRANSITION TO S50 ---
	IF (
		TRUE
	) THEN
	
		stepnumber:= 50;
		
	END_IF
		
		
		
	IF (stepnumber <> current_stepnumber) THEN
	
		// --- LAST SCAN ---
	
	
	END_IF
	

END_IF 

	
// Step 50
//___phase_example_Step_50_
//================================
// test a simple assignment with some BOOLS 
//================================	  

IF (stepnumber = 50) THEN

	
	IF (first_scan) THEN
	
		// --- FIRST SCAN ---
		

	ELSE
	
		// --- CONTINUOUS ---
		

		// Action: XV003_CMD = true
		XV003_CMD:= true;

		// Action: XV004_CMD = false
		XV004_CMD:= false;

	END_IF
	
	
	// --- TRANSITION TO S70 ---
	IF (
		TRUE
	) THEN
	
		stepnumber:= 70;
		
	END_IF
		
		
		
	IF (stepnumber <> current_stepnumber) THEN
	
		// --- LAST SCAN ---
	
	
	END_IF
	

END_IF 

	
// Step 70
//___phase_example_Step_70_
//================================
// test opening a valve 
//================================	  

IF (stepnumber = 70) THEN

	
	IF (first_scan) THEN
	
		// --- FIRST SCAN ---
		

	ELSE
	
		// --- CONTINUOUS ---
		

		// Action: open XV003
		XV003_CMD:= true;

	END_IF
	
	
	// --- TRANSITION TO S80 ---
	IF (
		TRUE
	) THEN
	
		stepnumber:= 80;
		
	END_IF
		
		
		
	IF (stepnumber <> current_stepnumber) THEN
	
		// --- LAST SCAN ---
	
	
	END_IF
	

END_IF 

	
// Step 80
//___phase_example_Step_80_
//================================
// test closing a valve 
//================================	  

IF (stepnumber = 80) THEN

	
	IF (first_scan) THEN
	
		// --- FIRST SCAN ---
		

	ELSE
	
		// --- CONTINUOUS ---
		

		// Action: close XV003
		XV003_CMD:= false;

	END_IF
	
	
	// --- TRANSITION TO S90 ---
	IF (
		TRUE
	) THEN
	
		stepnumber:= 90;
		
	END_IF
		
		
		
	IF (stepnumber <> current_stepnumber) THEN
	
		// --- LAST SCAN ---
	
	
	END_IF
	

END_IF 

	
// Step 90
//___phase_example_Step_90_
//================================
// test starting a motor 
//================================	  

IF (stepnumber = 90) THEN

	
	IF (first_scan) THEN
	
		// --- FIRST SCAN ---
		

	ELSE
	
		// --- CONTINUOUS ---
		

		// Action: start P001
		P001_ON:= true;

	END_IF
	
	
	// --- TRANSITION TO S100 ---
	IF (
		TRUE
	) THEN
	
		stepnumber:= 100;
		
	END_IF
		
		
		
	IF (stepnumber <> current_stepnumber) THEN
	
		// --- LAST SCAN ---
	
	
	END_IF
	

END_IF 

	
// Step 100
//___phase_example_Step_100_
//================================
// test stopping a motor 
//================================	  

IF (stepnumber = 100) THEN

	
	IF (first_scan) THEN
	
		// --- FIRST SCAN ---
		

	ELSE
	
		// --- CONTINUOUS ---
		

		// Action: stop P001
		P001_ON:= false;

	END_IF
	
	
	// --- TRANSITION TO S120 ---
	IF (
		TRUE
	) THEN
	
		stepnumber:= 120;
		
	END_IF
		
		
		
	IF (stepnumber <> current_stepnumber) THEN
	
		// --- LAST SCAN ---
	
	
	END_IF
	

END_IF 

	
// Step 120
//___phase_example_Step_120_
//================================
// test with some spaces and non-matching casing => should still work 
//================================	  

IF (stepnumber = 120) THEN

	
	IF (first_scan) THEN
	
		// --- FIRST SCAN ---
		

	ELSE
	
		// --- CONTINUOUS ---
		

		// Action: Open XV003
		XV003_CMD:= true;

	END_IF
	
	
	// --- TRANSITION TO S130 ---
	IF (
		TRUE
	) THEN
	
		stepnumber:= 130;
		
	END_IF
		
		
		
	IF (stepnumber <> current_stepnumber) THEN
	
		// --- LAST SCAN ---
	
	
	END_IF
	

END_IF 

	
// Step 130
//___phase_example_Step_130_
//================================
// test enumeration 
//================================	  

IF (stepnumber = 130) THEN

	
	IF (first_scan) THEN
	
		// --- FIRST SCAN ---
		

	ELSE
	
		// --- CONTINUOUS ---
		

		// Action: Destination = PF-I-02
		Destination:= 2;

	END_IF
	
	
	// --- TRANSITION TO S150 ---
	IF (
		TRUE
	) THEN
	
		stepnumber:= 150;
		
	END_IF
		
		
		
	IF (stepnumber <> current_stepnumber) THEN
	
		// --- LAST SCAN ---
	
	
	END_IF
	

END_IF 

	
// Step 150
//___phase_example_Step_150_
//================================
// test EM command 
//================================	  

IF (stepnumber = 150) THEN

	
	IF (first_scan) THEN
	
		// --- FIRST SCAN ---
		

	ELSE
	
		// --- CONTINUOUS ---
		

		// Action: EM_I_OUT = Pump_Fixed_Pressure
		EM_I_OUT.Command:= 2;

	END_IF
	
	
	// --- TRANSITION TO S170 ---
	IF (
		TRUE
	) THEN
	
		stepnumber:= 170;
		
	END_IF
		
		
		
	IF (stepnumber <> current_stepnumber) THEN
	
		// --- LAST SCAN ---
	
	
	END_IF
	

END_IF 

	
// Step 170
//___phase_example_Step_170_
//================================
// test some simple calculations 
//================================	  

IF (stepnumber = 170) THEN

	
	IF (first_scan) THEN
	
		// --- FIRST SCAN ---
		

	ELSE
	
		// --- CONTINUOUS ---
		

		// Action: xx = y * z
		xx:= y * z;

		// Action: rr = e / 2.0
		rr:= e / 2.0;

		// Action: g = h + ii
		g:= h + ii;

		// Action: j = k – mm
		j:= k - mm;

		// Action: n = o + 3.4
		n:= o + 3.4;

		// Action: pp = 7.3 / qq
		pp:= 7.3 / qq;

	END_IF
	
	
	// --- TRANSITION TO S180 ---
	IF (
		TRUE
	) THEN
	
		stepnumber:= 180;
		
	END_IF
		
		
		
	IF (stepnumber <> current_stepnumber) THEN
	
		// --- LAST SCAN ---
	
	
	END_IF
	

END_IF 

	
// Step 180
//___phase_example_Step_180_
//================================
// test complex calculations 
//================================	  

IF (stepnumber = 180) THEN

	
	IF (first_scan) THEN
	
		// --- FIRST SCAN ---
		

	ELSE
	
		// --- CONTINUOUS ---
		

		// Action: rr = (ss + tt) / u * v / (ww – xx + 1.34) + 2.3
		rr:= (ss + tt) / u * v / (ww - xx + 1.34) + 2.3;

		// Action: foo = bar + 1.0
		foo:= bar + 1.0;

		// Action: stoplevel = startlevel + setpoint – offset
		stoplevel:= startlevel + setpoint - offset;

	END_IF
	
	
	// --- TRANSITION TO S190 ---
	IF (
		TRUE
	) THEN
	
		stepnumber:= 190;
		
	END_IF
		
		
		
	IF (stepnumber <> current_stepnumber) THEN
	
		// --- LAST SCAN ---
	
	
	END_IF
	

END_IF 

	
// Step 190
//___phase_example_Step_190_
//================================
// add two REALs 
//================================	  

IF (stepnumber = 190) THEN

	
	IF (first_scan) THEN
	
		// --- FIRST SCAN ---
		

	ELSE
	
		// --- CONTINUOUS ---
		

		// Action: var1 = 3.0+2.0
		var1:= 3.0 + 2.0;

	END_IF
	
	
	// --- TRANSITION TO S200 ---
	IF (
		TRUE
	) THEN
	
		stepnumber:= 200;
		
	END_IF
		
		
		
	IF (stepnumber <> current_stepnumber) THEN
	
		// --- LAST SCAN ---
	
	
	END_IF
	

END_IF 

	
// Step 200
//___phase_example_Step_200_
//================================
// test first and last scan actions 
//================================	  

IF (stepnumber = 200) THEN

	
	IF (first_scan) THEN
	
		// --- FIRST SCAN ---
		

		// Action: xx = 1.0
		xx:= 1.0;

	ELSE
	
		// --- CONTINUOUS ---
		

		// Action: y = 2.0
		y:= 2.0;

	END_IF
	
	
	// --- TRANSITION TO S230 ---
	IF (
		TRUE
	) THEN
	
		stepnumber:= 230;
		
	END_IF
		
		
		
	IF (stepnumber <> current_stepnumber) THEN
	
		// --- LAST SCAN ---

		// Action: z = 3.0
		z:= 3.0;
	
	
	END_IF
	

END_IF 

	
// Step 230
//___phase_example_Step_230_
//================================
// test a transition with calculation 
//================================	  

IF (stepnumber = 230) THEN

	
	IF (first_scan) THEN
	
		// --- FIRST SCAN ---
		

	ELSE
	
		// --- CONTINUOUS ---
		

	END_IF
	
	
	// --- TRANSITION TO S250 ---
	IF (
		LT001_PV >= startlevel + setpoint - offset
	) THEN
	
		stepnumber:= 250;
		
	END_IF
		
		
		
	IF (stepnumber <> current_stepnumber) THEN
	
		// --- LAST SCAN ---
	
	
	END_IF
	

END_IF 

	
// Step 250
//___phase_example_Step_250_
//================================
// test natural language transition 
//================================	  

IF (stepnumber = 250) THEN

	
	IF (first_scan) THEN
	
		// --- FIRST SCAN ---
		

	ELSE
	
		// --- CONTINUOUS ---
		

	END_IF
	
	
	// --- TRANSITION TO S260 ---
	IF (
		P001_RUN
	) THEN
	
		stepnumber:= 260;
		
	END_IF
		
		
		
	IF (stepnumber <> current_stepnumber) THEN
	
		// --- LAST SCAN ---
	
	
	END_IF
	

END_IF 

	
// Step 260
//___phase_example_Step_260_
//================================
// test enumeration 
//================================	  

IF (stepnumber = 260) THEN

	
	IF (first_scan) THEN
	
		// --- FIRST SCAN ---
		

	ELSE
	
		// --- CONTINUOUS ---
		

	END_IF
	
	
	// --- TRANSITION TO S280 ---
	IF (
		Destination = 4
	) THEN
	
		stepnumber:= 280;
		
	END_IF
		
		
		
	IF (stepnumber <> current_stepnumber) THEN
	
		// --- LAST SCAN ---
	
	
	END_IF
	

END_IF 

	
// Step 280
//___phase_example_Step_280_
//================================
// test enumerated status of EM 
//================================	  

IF (stepnumber = 280) THEN

	
	IF (first_scan) THEN
	
		// --- FIRST SCAN ---
		

	ELSE
	
		// --- CONTINUOUS ---
		

	END_IF
	
	
	// --- TRANSITION TO S300 ---
	IF (
		EM_I_OUT.Status = 2
	) THEN
	
		stepnumber:= 300;
		
	END_IF
		
		
		
	IF (stepnumber <> current_stepnumber) THEN
	
		// --- LAST SCAN ---
	
	
	END_IF
	

END_IF 

	
// Step 300
//___phase_example_Step_300_
//================================
// test if primary suffixes are detected 
//================================	  

IF (stepnumber = 300) THEN

	
	IF (first_scan) THEN
	
		// --- FIRST SCAN ---
		

	ELSE
	
		// --- CONTINUOUS ---
		

	END_IF
	
	
	// --- TRANSITION TO S310 ---
	IF (
		2.0 * LT001_PV = (LT001_PV + LT001_PV - LT001_PV) * LT001_PV
	) THEN
	
		stepnumber:= 310;
		
	END_IF
		
		
		
	IF (stepnumber <> current_stepnumber) THEN
	
		// --- LAST SCAN ---
	
	
	END_IF
	

END_IF 

	
// Step 310
//___phase_example_Step_310_
//================================
// test primary suffixes in action side 
//================================	  

IF (stepnumber = 310) THEN

	
	IF (first_scan) THEN
	
		// --- FIRST SCAN ---
		

	ELSE
	
		// --- CONTINUOUS ---
		

		// Action: test1 = (LT001 + LT001 – LT001) * LT001
		test1:= (LT001_PV + LT001_PV - LT001_PV) * LT001_PV;

		// Action: test2 = LT002
		test2:= LT002_PV;

	END_IF
	
	
	// --- TRANSITION TO S320 ---
	IF (
		TRUE
	) THEN
	
		stepnumber:= 320;
		
	END_IF
		
		
		
	IF (stepnumber <> current_stepnumber) THEN
	
		// --- LAST SCAN ---
	
	
	END_IF
	

END_IF 

	
// Step 320
//___phase_example_Step_320_
//================================
// test with AND in front 
//================================	  

IF (stepnumber = 320) THEN

	
	IF (first_scan) THEN
	
		// --- FIRST SCAN ---
		

	ELSE
	
		// --- CONTINUOUS ---
		

	END_IF
	
	
	// --- TRANSITION TO S330 ---
	IF (
		XV003_OPN
	) THEN
	
		stepnumber:= 330;
		
	END_IF
		
		
		
	IF (stepnumber <> current_stepnumber) THEN
	
		// --- LAST SCAN ---
	
	
	END_IF
	

END_IF 

	
// Step 330
//___phase_example_Step_330_
//================================
// test multiple conditions without explicit logic 
//================================	  

IF (stepnumber = 330) THEN

	
	IF (first_scan) THEN
	
		// --- FIRST SCAN ---
		

	ELSE
	
		// --- CONTINUOUS ---
		

	END_IF
	
	
	// --- TRANSITION TO S340 ---
	IF (
		XV003_OPN
		AND XV004_OPN
	) THEN
	
		stepnumber:= 340;
		
	END_IF
		
		
		
	IF (stepnumber <> current_stepnumber) THEN
	
		// --- LAST SCAN ---
	
	
	END_IF
	

END_IF 

	
// Step 340
//___phase_example_Step_340_
//================================
// test multiple conditions with logic 
//================================	  

IF (stepnumber = 340) THEN

	
	IF (first_scan) THEN
	
		// --- FIRST SCAN ---
		

	ELSE
	
		// --- CONTINUOUS ---
		

	END_IF
	
	
	// --- TRANSITION TO S350 ---
	IF (
		XV003_OPN
		AND XV004_OPN
	) THEN
	
		stepnumber:= 350;
		
	END_IF
		
		
		
	IF (stepnumber <> current_stepnumber) THEN
	
		// --- LAST SCAN ---
	
	
	END_IF
	

END_IF 

	
// Step 350
//___phase_example_Step_350_
//================================
// test OR-logic 
//================================	  

IF (stepnumber = 350) THEN

	
	IF (first_scan) THEN
	
		// --- FIRST SCAN ---
		

	ELSE
	
		// --- CONTINUOUS ---
		

	END_IF
	
	
	// --- TRANSITION TO S360 ---
	IF (
		XV003_OPN
		OR XV004_OPN
	) THEN
	
		stepnumber:= 360;
		
	END_IF
		
		
		
	IF (stepnumber <> current_stepnumber) THEN
	
		// --- LAST SCAN ---
	
	
	END_IF
	

END_IF 

	
// Step 360
//___phase_example_Step_360_
//================================
// test combined logic 
//================================	  

IF (stepnumber = 360) THEN

	
	IF (first_scan) THEN
	
		// --- FIRST SCAN ---
		

	ELSE
	
		// --- CONTINUOUS ---
		

	END_IF
	
	
	// --- TRANSITION TO S370 ---
	IF (
		XV005_OPN
		AND( 
			XV003_OPN
			OR XV004_OPN
		) 
	) THEN
	
		stepnumber:= 370;
		
	END_IF
		
		
		
	IF (stepnumber <> current_stepnumber) THEN
	
		// --- LAST SCAN ---
	
	
	END_IF
	

END_IF 

	
// Step 370
//___phase_example_Step_370_
//================================
// test improved readability 
//================================	  

IF (stepnumber = 370) THEN

	
	IF (first_scan) THEN
	
		// --- FIRST SCAN ---
		

	ELSE
	
		// --- CONTINUOUS ---
		

	END_IF
	
	
	// --- TRANSITION TO S420 ---
	IF (
		XV005_OPN
		AND( 
			XV003_OPN
			OR XV004_OPN
		) 
	) THEN
	
		stepnumber:= 420;
		
	END_IF
		
		
		
	IF (stepnumber <> current_stepnumber) THEN
	
		// --- LAST SCAN ---
	
	
	END_IF
	

END_IF 

	
// Step 420
//___phase_example_Step_420_
//================================
// test first line without logic and rest with AND 
//================================	  

IF (stepnumber = 420) THEN

	
	IF (first_scan) THEN
	
		// --- FIRST SCAN ---
		

	ELSE
	
		// --- CONTINUOUS ---
		

	END_IF
	
	
	// --- TRANSITION TO S430 ---
	IF (
		XV003_OPN
		AND XV004_OPN
		AND XV005_OPN
	) THEN
	
		stepnumber:= 430;
		
	END_IF
		
		
		
	IF (stepnumber <> current_stepnumber) THEN
	
		// --- LAST SCAN ---
	
	
	END_IF
	

END_IF 

	
// Step 430
//___phase_example_Step_430_
//================================
// test first line without logic and rest with OR 
//================================	  

IF (stepnumber = 430) THEN

	
	IF (first_scan) THEN
	
		// --- FIRST SCAN ---
		

	ELSE
	
		// --- CONTINUOUS ---
		

	END_IF
	
	
	// --- TRANSITION TO S440 ---
	IF (
		XV003_OPN
		OR XV004_OPN
		OR XV005_OPN
	) THEN
	
		stepnumber:= 440;
		
	END_IF
		
		
		
	IF (stepnumber <> current_stepnumber) THEN
	
		// --- LAST SCAN ---
	
	
	END_IF
	

END_IF 

	
// Step 440
//___phase_example_Step_440_
//================================
// test button 
//================================	  

IF (stepnumber = 440) THEN

	
	IF (first_scan) THEN
	
		// --- FIRST SCAN ---
		

	ELSE
	
		// --- CONTINUOUS ---
		

		// Action: show button_1
		button_1_visible:= true;

		// Action: select text with ID 16: continue
		button_1_text:= 16;

	END_IF
	
	
	// --- TRANSITION TO S450 ---
	IF (
		button_1_pushed
	) THEN
	
		stepnumber:= 450;
		
	END_IF
		
		
		
	IF (stepnumber <> current_stepnumber) THEN
	
		// --- LAST SCAN ---

		// Action: hide button_1
		button_1_visible:= false;
	
	
	END_IF
	

END_IF 

	
// Step 450
//___phase_example_Step_450_
//================================
// test button with capital => no problem, the button is case insensitive 
//================================	  

IF (stepnumber = 450) THEN

	
	IF (first_scan) THEN
	
		// --- FIRST SCAN ---
		

	ELSE
	
		// --- CONTINUOUS ---
		

		// Action: show button_1
		button_1_visible:= true;

		// Action: select text with ID 17: ok
		button_1_text:= 17;

	END_IF
	
	
	// --- TRANSITION TO S460 ---
	IF (
		button_1_pushed
	) THEN
	
		stepnumber:= 460;
		
	END_IF
		
		
		
	IF (stepnumber <> current_stepnumber) THEN
	
		// --- LAST SCAN ---

		// Action: hide button_1
		button_1_visible:= false;
	
	
	END_IF
	

END_IF 

	
// Step 460
//___phase_example_Step_460_
//================================
// test button without opening quotation marks => no problem, any marks are just removed 
//================================	  

IF (stepnumber = 460) THEN

	
	IF (first_scan) THEN
	
		// --- FIRST SCAN ---
		

	ELSE
	
		// --- CONTINUOUS ---
		

		// Action: show button_1
		button_1_visible:= true;

		// Action: select text with ID 18: cancel
		button_1_text:= 18;

	END_IF
	
	
	// --- TRANSITION TO S470 ---
	IF (
		button_1_pushed
	) THEN
	
		stepnumber:= 470;
		
	END_IF
		
		
		
	IF (stepnumber <> current_stepnumber) THEN
	
		// --- LAST SCAN ---

		// Action: hide button_1
		button_1_visible:= false;
	
	
	END_IF
	

END_IF 

	
// Step 470
//___phase_example_Step_470_
//================================
// test button without closing quotation marks => no problem, any marks are just removed 
//================================	  

IF (stepnumber = 470) THEN

	
	IF (first_scan) THEN
	
		// --- FIRST SCAN ---
		

	ELSE
	
		// --- CONTINUOUS ---
		

		// Action: show button_1
		button_1_visible:= true;

		// Action: select text with ID 19: go back
		button_1_text:= 19;

	END_IF
	
	
	// --- TRANSITION TO S480 ---
	IF (
		button_1_pushed
	) THEN
	
		stepnumber:= 480;
		
	END_IF
		
		
		
	IF (stepnumber <> current_stepnumber) THEN
	
		// --- LAST SCAN ---

		// Action: hide button_1
		button_1_visible:= false;
	
	
	END_IF
	

END_IF 

	
// Step 480
//___phase_example_Step_480_
//================================
// test 3 buttons 
//================================	  

IF (stepnumber = 480) THEN

	
	IF (first_scan) THEN
	
		// --- FIRST SCAN ---
		

	ELSE
	
		// --- CONTINUOUS ---
		

		// Action: show button_1
		button_1_visible:= true;

		// Action: select text with ID 16: continue
		button_1_text:= 16;

		// Action: show button_2
		button_2_visible:= true;

		// Action: select text with ID 18: cancel
		button_2_text:= 18;

		// Action: show button_3
		button_3_visible:= true;

		// Action: select text with ID 19: go back
		button_3_text:= 19;

	END_IF
	
	
	// --- TRANSITION TO S490 ---
	IF (
		button_1_pushed
		AND button_2_pushed
		AND button_3_pushed
	) THEN
	
		stepnumber:= 490;
		
	END_IF
		
		
		
	IF (stepnumber <> current_stepnumber) THEN
	
		// --- LAST SCAN ---

		// Action: hide button_1
		button_1_visible:= false;

		// Action: hide button_2
		button_2_visible:= false;

		// Action: hide button_3
		button_3_visible:= false;
	
	
	END_IF
	

END_IF 

	
// Step 490
//___phase_example_Step_490_
//================================
// test 4 buttons => not foreseen in the template, so should log an error 
//================================	  

IF (stepnumber = 490) THEN

	
	IF (first_scan) THEN
	
		// --- FIRST SCAN ---
		

	ELSE
	
		// --- CONTINUOUS ---
		

		// Action: show button_1
		button_1_visible:= true;

		// Action: select text with ID 16: continue
		button_1_text:= 16;

		// Action: show button_2
		button_2_visible:= true;

		// Action: select text with ID 18: cancel
		button_2_text:= 18;

		// Action: show button_3
		button_3_visible:= true;

		// Action: select text with ID 19: go back
		button_3_text:= 19;

	END_IF
	
	
	// --- TRANSITION TO S510 ---
	IF (
		button_1_pushed
		AND button_2_pushed
		AND button_3_pushed
	) THEN
	
		stepnumber:= 510;
		
	END_IF
		
		
		
	IF (stepnumber <> current_stepnumber) THEN
	
		// --- LAST SCAN ---

		// Action: hide button_1
		button_1_visible:= false;

		// Action: hide button_2
		button_2_visible:= false;

		// Action: hide button_3
		button_3_visible:= false;
	
	
	END_IF
	

END_IF 

	
// Step 510
//___phase_example_Step_510_
//================================
// test message 
//================================	  

IF (stepnumber = 510) THEN

	
	IF (first_scan) THEN
	
		// --- FIRST SCAN ---
		

	ELSE
	
		// --- CONTINUOUS ---
		

		// Action: message “add the manual ingredients”
		message:= 21;

	END_IF
	
	
	// --- TRANSITION TO S520 ---
	IF (
		TRUE
	) THEN
	
		stepnumber:= 520;
		
	END_IF
		
		
		
	IF (stepnumber <> current_stepnumber) THEN
	
		// --- LAST SCAN ---

		// Action: clear message
		message:= 0;
	
	
	END_IF
	

END_IF 

	
// Step 520
//___phase_example_Step_520_
//================================
// test falseword with two words in transition 
//================================	  

IF (stepnumber = 520) THEN

	
	IF (first_scan) THEN
	
		// --- FIRST SCAN ---
		

	ELSE
	
		// --- CONTINUOUS ---
		

	END_IF
	
	
	// --- TRANSITION TO S530 ---
	IF (
		XV003_OPN
	) THEN
	
		stepnumber:= 530;
		
	END_IF
		
		
		
	IF (stepnumber <> current_stepnumber) THEN
	
		// --- LAST SCAN ---
	
	
	END_IF
	

END_IF 

	
// Step 530
//___phase_example_Step_530_
//================================
// test trueword with multiple words in action 
//================================	  

IF (stepnumber = 530) THEN

	
	IF (first_scan) THEN
	
		// --- FIRST SCAN ---
		

	ELSE
	
		// --- CONTINUOUS ---
		

		// Action: move to open position XV003
		XV003_CMD:= true;

	END_IF
	
	
	// --- TRANSITION TO S540 ---
	IF (
		TRUE
	) THEN
	
		stepnumber:= 540;
		
	END_IF
		
		
		
	IF (stepnumber <> current_stepnumber) THEN
	
		// --- LAST SCAN ---
	
	
	END_IF
	

END_IF 

	
// Step 540
//___phase_example_Step_540_
//================================
// test putting controller in auto with pulseword 
//================================	  

IF (stepnumber = 540) THEN

	
	IF (first_scan) THEN
	
		// --- FIRST SCAN ---
		

	ELSE
	
		// --- CONTINUOUS ---
		

		// Action: FIC001 auto
		FIC001_AUT:= true;

	END_IF
	
	
	// --- TRANSITION TO S550 ---
	IF (
		TRUE
	) THEN
	
		stepnumber:= 550;
		
	END_IF
		
		
		
	IF (stepnumber <> current_stepnumber) THEN
	
		// --- LAST SCAN ---
	
	
	END_IF
	

END_IF 

	
// Step 550
//___phase_example_Step_550_
//================================
// test putting controller in auto with pulseword consisting of multiple words 
//================================	  

IF (stepnumber = 550) THEN

	
	IF (first_scan) THEN
	
		// --- FIRST SCAN ---
		

	ELSE
	
		// --- CONTINUOUS ---
		

		// Action: FIC001 switch to auto
		FIC001_AUT:= true;

	END_IF
	
	
	// --- TRANSITION TO S560 ---
	IF (
		TRUE
	) THEN
	
		stepnumber:= 560;
		
	END_IF
		
		
		
	IF (stepnumber <> current_stepnumber) THEN
	
		// --- LAST SCAN ---
	
	
	END_IF
	

END_IF 

	
// Step 560
//___phase_example_Step_560_
//================================
// test with pulseword in front 
//================================	  

IF (stepnumber = 560) THEN

	
	IF (first_scan) THEN
	
		// --- FIRST SCAN ---
		

	ELSE
	
		// --- CONTINUOUS ---
		

		// Action: auto FIC001
		FIC001_AUT:= true;

	END_IF
	
	
	// --- TRANSITION TO S570 ---
	IF (
		TRUE
	) THEN
	
		stepnumber:= 570;
		
	END_IF
		
		
		
	IF (stepnumber <> current_stepnumber) THEN
	
		// --- LAST SCAN ---
	
	
	END_IF
	

END_IF 

	
// Step 570
//___phase_example_Step_570_
//================================
// test with pulseword in front 
//================================	  

IF (stepnumber = 570) THEN

	
	IF (first_scan) THEN
	
		// --- FIRST SCAN ---
		

	ELSE
	
		// --- CONTINUOUS ---
		

		// Action: switch to auto FIC001
		FIC001_AUT:= true;

	END_IF
	
	
	// --- TRANSITION TO S580 ---
	IF (
		TRUE
	) THEN
	
		stepnumber:= 580;
		
	END_IF
		
		
		
	IF (stepnumber <> current_stepnumber) THEN
	
		// --- LAST SCAN ---
	
	
	END_IF
	

END_IF 

	
// Step 580
//___phase_example_Step_580_
//================================
// test steptime in s 
//================================	  

IF (stepnumber = 580) THEN

	
	IF (first_scan) THEN
	
		// --- FIRST SCAN ---
		

	ELSE
	
		// --- CONTINUOUS ---
		

	END_IF
	
	
	// --- TRANSITION TO S590 ---
	IF (
		steptime_s > 2.0
	) THEN
	
		stepnumber:= 590;
		
	END_IF
		
		
		
	IF (stepnumber <> current_stepnumber) THEN
	
		// --- LAST SCAN ---
	
	
	END_IF
	

END_IF 

	
// Step 590
//___phase_example_Step_590_
//================================
// test steptime in m 
//================================	  

IF (stepnumber = 590) THEN

	
	IF (first_scan) THEN
	
		// --- FIRST SCAN ---
		

	ELSE
	
		// --- CONTINUOUS ---
		

	END_IF
	
	
	// --- TRANSITION TO S600 ---
	IF (
		steptime_m > 1.50
	) THEN
	
		stepnumber:= 600;
		
	END_IF
		
		
		
	IF (stepnumber <> current_stepnumber) THEN
	
		// --- LAST SCAN ---
	
	
	END_IF
	

END_IF 

	
// Step 600
//___phase_example_Step_600_
//================================
// test steptime in h 
//================================	  

IF (stepnumber = 600) THEN

	
	IF (first_scan) THEN
	
		// --- FIRST SCAN ---
		

	ELSE
	
		// --- CONTINUOUS ---
		

	END_IF
	
	
	// --- TRANSITION TO S610 ---
	IF (
		steptime_h > 4.3
	) THEN
	
		stepnumber:= 610;
		
	END_IF
		
		
		
	IF (stepnumber <> current_stepnumber) THEN
	
		// --- LAST SCAN ---
	
	
	END_IF
	

END_IF 

	
// Step 610
//___phase_example_Step_610_
//================================
// test steptime with unit separated by space => still works (because it takes the last character) 
//================================	  

IF (stepnumber = 610) THEN

	
	IF (first_scan) THEN
	
		// --- FIRST SCAN ---
		

	ELSE
	
		// --- CONTINUOUS ---
		

	END_IF
	
	
	// --- TRANSITION TO S640 ---
	IF (
		steptime_m > 1.50
	) THEN
	
		stepnumber:= 640;
		
	END_IF
		
		
		
	IF (stepnumber <> current_stepnumber) THEN
	
		// --- LAST SCAN ---
	
	
	END_IF
	

END_IF 

	
// Step 640
//___phase_example_Step_640_
//================================
// test steptime with variable with unit 
//================================	  

IF (stepnumber = 640) THEN

	
	IF (first_scan) THEN
	
		// --- FIRST SCAN ---
		

	ELSE
	
		// --- CONTINUOUS ---
		

	END_IF
	
	
	// --- TRANSITION TO S650 ---
	IF (
		steptime_h > timesetting
	) THEN
	
		stepnumber:= 650;
		
	END_IF
		
		
		
	IF (stepnumber <> current_stepnumber) THEN
	
		// --- LAST SCAN ---
	
	
	END_IF
	

END_IF 

	
// Step 650
//___phase_example_Step_650_
//================================
// reset a timer 
//================================	  

IF (stepnumber = 650) THEN

	
	IF (first_scan) THEN
	
		// --- FIRST SCAN ---
		

	ELSE
	
		// --- CONTINUOUS ---
		

		// Action: reset timer_dosing
		timer_dosing_s:= 0.0;

	END_IF
	
	
	// --- TRANSITION TO S660 ---
	IF (
		TRUE
	) THEN
	
		stepnumber:= 660;
		
	END_IF
		
		
		
	IF (stepnumber <> current_stepnumber) THEN
	
		// --- LAST SCAN ---
	
	
	END_IF
	

END_IF 

	
// Step 660
//___phase_example_Step_660_
//================================
// start a timer 
//================================	  

IF (stepnumber = 660) THEN

	
	IF (first_scan) THEN
	
		// --- FIRST SCAN ---
		

	ELSE
	
		// --- CONTINUOUS ---
		

		// Action: start timer_mixing
		timer_mixing_pause:= false;

	END_IF
	
	
	// --- TRANSITION TO S670 ---
	IF (
		TRUE
	) THEN
	
		stepnumber:= 670;
		
	END_IF
		
		
		
	IF (stepnumber <> current_stepnumber) THEN
	
		// --- LAST SCAN ---
	
	
	END_IF
	

END_IF 

	
// Step 670
//___phase_example_Step_670_
//================================
// pause a timer 
//================================	  

IF (stepnumber = 670) THEN

	
	IF (first_scan) THEN
	
		// --- FIRST SCAN ---
		

	ELSE
	
		// --- CONTINUOUS ---
		

		// Action: pause timer_circulation
		timer_circulation_pause:= true;

	END_IF
	
	
	// --- TRANSITION TO S680 ---
	IF (
		TRUE
	) THEN
	
		stepnumber:= 680;
		
	END_IF
		
		
		
	IF (stepnumber <> current_stepnumber) THEN
	
		// --- LAST SCAN ---
	
	
	END_IF
	

END_IF 

	
// Step 680
//___phase_example_Step_680_
//================================
// test timer in m 
//================================	  

IF (stepnumber = 680) THEN

	
	IF (first_scan) THEN
	
		// --- FIRST SCAN ---
		

	ELSE
	
		// --- CONTINUOUS ---
		

	END_IF
	
	
	// --- TRANSITION TO S690 ---
	IF (
		timer_dosing_m >= 5.2
	) THEN
	
		stepnumber:= 690;
		
	END_IF
		
		
		
	IF (stepnumber <> current_stepnumber) THEN
	
		// --- LAST SCAN ---
	
	
	END_IF
	

END_IF 

	
// Step 690
//___phase_example_Step_690_
//================================
// test timer with variable with unit 
//================================	  

IF (stepnumber = 690) THEN

	
	IF (first_scan) THEN
	
		// --- FIRST SCAN ---
		

	ELSE
	
		// --- CONTINUOUS ---
		

	END_IF
	
	
	// --- TRANSITION TO S700 ---
	IF (
		timer_circulation_h < timesetting
	) THEN
	
		stepnumber:= 700;
		
	END_IF
		
		
		
	IF (stepnumber <> current_stepnumber) THEN
	
		// --- LAST SCAN ---
	
	
	END_IF
	

END_IF 

	
// Step 700
//___phase_example_Step_700_
//================================
// test putting a controller in manual 
//================================	  

IF (stepnumber = 700) THEN

	
	IF (first_scan) THEN
	
		// --- FIRST SCAN ---
		

	ELSE
	
		// --- CONTINUOUS ---
		

		// Action: FIC001 manual
		FIC001_AUT:= false;

	END_IF
	
	
	// --- TRANSITION TO S710 ---
	IF (
		TRUE
	) THEN
	
		stepnumber:= 710;
		
	END_IF
		
		
		
	IF (stepnumber <> current_stepnumber) THEN
	
		// --- LAST SCAN ---
	
	
	END_IF
	

END_IF 

	
// Step 710
//___phase_example_Step_710_
//================================
// test putting a controller in manual while changing the output value 
//================================	  

IF (stepnumber = 710) THEN

	
	IF (first_scan) THEN
	
		// --- FIRST SCAN ---
		

		// Action: FIC001_VAL_OUT = 20.0
		FIC001_VAL_OUT:= 20.0;

		// Action: FIC001_SET_OUT = true
		FIC001_SET_OUT:= true;

	ELSE
	
		// --- CONTINUOUS ---
		

		// Action: FIC001 manual 20.0
		FIC001_AUT:= false;

		// Action: FIC001_SET_OUT = false
		FIC001_SET_OUT:= false;

	END_IF
	
	
	// --- TRANSITION TO S720 ---
	IF (
		TRUE
	) THEN
	
		stepnumber:= 720;
		
	END_IF
		
		
		
	IF (stepnumber <> current_stepnumber) THEN
	
		// --- LAST SCAN ---
	
	
	END_IF
	

END_IF 

	
// Step 720
//___phase_example_Step_720_
//================================
// test putting a controller in manual while changing the output value that has a unit 
//================================	  

IF (stepnumber = 720) THEN

	
	IF (first_scan) THEN
	
		// --- FIRST SCAN ---
		

		// Action: FIC001_VAL_OUT = 20.0
		FIC001_VAL_OUT:= 20.0;

		// Action: FIC001_SET_OUT = true
		FIC001_SET_OUT:= true;

	ELSE
	
		// --- CONTINUOUS ---
		

		// Action: FIC001 manual 20.0 Hz
		FIC001_AUT:= false;

		// Action: FIC001_SET_OUT = false
		FIC001_SET_OUT:= false;

	END_IF
	
	
	// --- TRANSITION TO S730 ---
	IF (
		TRUE
	) THEN
	
		stepnumber:= 730;
		
	END_IF
		
		
		
	IF (stepnumber <> current_stepnumber) THEN
	
		// --- LAST SCAN ---
	
	
	END_IF
	

END_IF 

	
// Step 730
//___phase_example_Step_730_
//================================
// without space 
//================================	  

IF (stepnumber = 730) THEN

	
	IF (first_scan) THEN
	
		// --- FIRST SCAN ---
		

		// Action: FIC001_VAL_OUT = 20.0
		FIC001_VAL_OUT:= 20.0;

		// Action: FIC001_SET_OUT = true
		FIC001_SET_OUT:= true;

	ELSE
	
		// --- CONTINUOUS ---
		

		// Action: FIC001 manual 20.0Hz
		FIC001_AUT:= false;

		// Action: FIC001_SET_OUT = false
		FIC001_SET_OUT:= false;

	END_IF
	
	
	// --- TRANSITION TO S740 ---
	IF (
		TRUE
	) THEN
	
		stepnumber:= 740;
		
	END_IF
		
		
		
	IF (stepnumber <> current_stepnumber) THEN
	
		// --- LAST SCAN ---
	
	
	END_IF
	

END_IF 

	
// Step 740
//___phase_example_Step_740_
//================================
// put PID controller in auto 
//================================	  

IF (stepnumber = 740) THEN

	
	IF (first_scan) THEN
	
		// --- FIRST SCAN ---
		

	ELSE
	
		// --- CONTINUOUS ---
		

		// Action: FIC001 auto
		FIC001_AUT:= true;

	END_IF
	
	
	// --- TRANSITION TO S750 ---
	IF (
		TRUE
	) THEN
	
		stepnumber:= 750;
		
	END_IF
		
		
		
	IF (stepnumber <> current_stepnumber) THEN
	
		// --- LAST SCAN ---
	
	
	END_IF
	

END_IF 

	
// Step 750
//___phase_example_Step_750_
//================================
// auto with setpoint 
//================================	  

IF (stepnumber = 750) THEN

	
	IF (first_scan) THEN
	
		// --- FIRST SCAN ---
		

		// Action: FIC001_SP = 80.0
		FIC001_SP:= 80.0;

		// Action: FIC001_SET_SP = true
		FIC001_SET_SP:= true;

	ELSE
	
		// --- CONTINUOUS ---
		

		// Action: FIC001 auto 80.0%
		FIC001_AUT:= true;

		// Action: FIC001_SET_SP = false
		FIC001_SET_SP:= false;

	END_IF
	
	
	// --- TRANSITION TO S760 ---
	IF (
		TRUE
	) THEN
	
		stepnumber:= 760;
		
	END_IF
		
		
		
	IF (stepnumber <> current_stepnumber) THEN
	
		// --- LAST SCAN ---
	
	
	END_IF
	

END_IF 

	
// Step 760
//___phase_example_Step_760_
//================================
// internal mode 
//================================	  

IF (stepnumber = 760) THEN

	
	IF (first_scan) THEN
	
		// --- FIRST SCAN ---
		

	ELSE
	
		// --- CONTINUOUS ---
		

		// Action: FIC001 internal
		FIC001_EXT:= false;

	END_IF
	
	
	// --- TRANSITION TO S770 ---
	IF (
		TRUE
	) THEN
	
		stepnumber:= 770;
		
	END_IF
		
		
		
	IF (stepnumber <> current_stepnumber) THEN
	
		// --- LAST SCAN ---
	
	
	END_IF
	

END_IF 

	
// Step 770
//___phase_example_Step_770_
//================================
// internal mode with value 
//================================	  

IF (stepnumber = 770) THEN

	
	IF (first_scan) THEN
	
		// --- FIRST SCAN ---
		

		// Action: FIC001_SP = 80.0
		FIC001_SP:= 80.0;

		// Action: FIC001_SET_SP = true
		FIC001_SET_SP:= true;

	ELSE
	
		// --- CONTINUOUS ---
		

		// Action: FIC001 internal 80.0
		FIC001_EXT:= false;

		// Action: FIC001_SET_SP = false
		FIC001_SET_SP:= false;

	END_IF
	
	
	// --- TRANSITION TO S780 ---
	IF (
		TRUE
	) THEN
	
		stepnumber:= 780;
		
	END_IF
		
		
		
	IF (stepnumber <> current_stepnumber) THEN
	
		// --- LAST SCAN ---
	
	
	END_IF
	

END_IF 

	
// Step 780
//___phase_example_Step_780_
//================================
// value with unit 
//================================	  

IF (stepnumber = 780) THEN

	
	IF (first_scan) THEN
	
		// --- FIRST SCAN ---
		

		// Action: FIC001_SP = 80.0
		FIC001_SP:= 80.0;

		// Action: FIC001_SET_SP = true
		FIC001_SET_SP:= true;

	ELSE
	
		// --- CONTINUOUS ---
		

		// Action: FIC001 internal 80.0 %
		FIC001_EXT:= false;

		// Action: FIC001_SET_SP = false
		FIC001_SET_SP:= false;

	END_IF
	
	
	// --- TRANSITION TO S790 ---
	IF (
		TRUE
	) THEN
	
		stepnumber:= 790;
		
	END_IF
		
		
		
	IF (stepnumber <> current_stepnumber) THEN
	
		// --- LAST SCAN ---
	
	
	END_IF
	

END_IF 

	
// Step 790
//___phase_example_Step_790_
//================================
// without space 
//================================	  

IF (stepnumber = 790) THEN

	
	IF (first_scan) THEN
	
		// --- FIRST SCAN ---
		

		// Action: FIC001_SP = 80.0
		FIC001_SP:= 80.0;

		// Action: FIC001_SET_SP = true
		FIC001_SET_SP:= true;

	ELSE
	
		// --- CONTINUOUS ---
		

		// Action: FIC001 internal80.0%
		FIC001_EXT:= false;

		// Action: FIC001_SET_SP = false
		FIC001_SET_SP:= false;

	END_IF
	
	
	// --- TRANSITION TO S810 ---
	IF (
		TRUE
	) THEN
	
		stepnumber:= 810;
		
	END_IF
		
		
		
	IF (stepnumber <> current_stepnumber) THEN
	
		// --- LAST SCAN ---
	
	
	END_IF
	

END_IF 

	
// Step 810
//___phase_example_Step_810_
//================================
// external mode 
//================================	  

IF (stepnumber = 810) THEN

	
	IF (first_scan) THEN
	
		// --- FIRST SCAN ---
		

	ELSE
	
		// --- CONTINUOUS ---
		

		// Action: FIC001 external
		FIC001_EXT:= true;

	END_IF
	
	
	// --- TRANSITION TO S820 ---
	IF (
		TRUE
	) THEN
	
		stepnumber:= 820;
		
	END_IF
		
		
		
	IF (stepnumber <> current_stepnumber) THEN
	
		// --- LAST SCAN ---
	
	
	END_IF
	

END_IF 

	
// Step 820
//___phase_example_Step_820_
//================================
// test direct access to a CM instance in dot-format in the assignment => should convert to suffix 
//================================	  

IF (stepnumber = 820) THEN

	
	IF (first_scan) THEN
	
		// --- FIRST SCAN ---
		

	ELSE
	
		// --- CONTINUOUS ---
		

		// Action: XV008.AUT_OP = true
		XV008_CMD:= true;

	END_IF
	
	
	// --- TRANSITION TO S830 ---
	IF (
		TRUE
	) THEN
	
		stepnumber:= 830;
		
	END_IF
		
		
		
	IF (stepnumber <> current_stepnumber) THEN
	
		// --- LAST SCAN ---
	
	
	END_IF
	

END_IF 

	
// Step 830
//___phase_example_Step_830_
//================================
// test direct access to a CM in dot-notation in the evaluation => should convert to suffix 
//================================	  

IF (stepnumber = 830) THEN

	
	IF (first_scan) THEN
	
		// --- FIRST SCAN ---
		

	ELSE
	
		// --- CONTINUOUS ---
		

	END_IF
	
	
	// --- TRANSITION TO S840 ---
	IF (
		XV008_OPN = true
	) THEN
	
		stepnumber:= 840;
		
	END_IF
		
		
		
	IF (stepnumber <> current_stepnumber) THEN
	
		// --- LAST SCAN ---
	
	
	END_IF
	

END_IF 

	
// Step 840
//___phase_example_Step_840_
//================================
// test dot-format to Linked CM in assignment => should convert to suffix 
//================================	  

IF (stepnumber = 840) THEN

	
	IF (first_scan) THEN
	
		// --- FIRST SCAN ---
		

	ELSE
	
		// --- CONTINUOUS ---
		

		// Action: XV003.AUT_OP = true
		XV003_CMD:= true;

	END_IF
	
	
	// --- TRANSITION TO S850 ---
	IF (
		TRUE
	) THEN
	
		stepnumber:= 850;
		
	END_IF
		
		
		
	IF (stepnumber <> current_stepnumber) THEN
	
		// --- LAST SCAN ---
	
	
	END_IF
	

END_IF 

	
// Step 850
//___phase_example_Step_850_
//================================
// test dot-format from Linked CM in evaluation =>should convert to suffix 
//================================	  

IF (stepnumber = 850) THEN

	
	IF (first_scan) THEN
	
		// --- FIRST SCAN ---
		

	ELSE
	
		// --- CONTINUOUS ---
		

	END_IF
	
	
	// --- TRANSITION TO S860 ---
	IF (
		XV003_OPN = true
	) THEN
	
		stepnumber:= 860;
		
	END_IF
		
		
		
	IF (stepnumber <> current_stepnumber) THEN
	
		// --- LAST SCAN ---
	
	
	END_IF
	

END_IF 

	
// Step 860
//___phase_example_Step_860_
//================================
// test direct access to an EM instance in dot-format in the assignment => should stay in dot-format 
//================================	  

IF (stepnumber = 860) THEN

	
	IF (first_scan) THEN
	
		// --- FIRST SCAN ---
		

	ELSE
	
		// --- CONTINUOUS ---
		

		// Action: EM_Instance_4.Pressure_SP  = 4.2
		EM_Instance_4.Pressure_SP:= 4.2;

	END_IF
	
	
	// --- TRANSITION TO S870 ---
	IF (
		TRUE
	) THEN
	
		stepnumber:= 870;
		
	END_IF
		
		
		
	IF (stepnumber <> current_stepnumber) THEN
	
		// --- LAST SCAN ---
	
	
	END_IF
	

END_IF 

	
// Step 870
//___phase_example_Step_870_
//================================
// test direct access to a EM in dot-notation in the evaluation => should stay in dot-format 
//================================	  

IF (stepnumber = 870) THEN

	
	IF (first_scan) THEN
	
		// --- FIRST SCAN ---
		

	ELSE
	
		// --- CONTINUOUS ---
		

	END_IF
	
	
	// --- TRANSITION TO S880 ---
	IF (
		EM_Instance_4.Level >= 50.0
	) THEN
	
		stepnumber:= 880;
		
	END_IF
		
		
		
	IF (stepnumber <> current_stepnumber) THEN
	
		// --- LAST SCAN ---
	
	
	END_IF
	

END_IF 

	
// Step 880
//___phase_example_Step_880_
//================================
// test dot-format to Linked EM in assignment => should stay in dot-format 
//================================	  

IF (stepnumber = 880) THEN

	
	IF (first_scan) THEN
	
		// --- FIRST SCAN ---
		

	ELSE
	
		// --- CONTINUOUS ---
		

		// Action: Some_Dyn_EM.Pressure_SP  = 4.2
		Some_Dyn_EM.Pressure_SP:= 4.2;

	END_IF
	
	
	// --- TRANSITION TO S890 ---
	IF (
		TRUE
	) THEN
	
		stepnumber:= 890;
		
	END_IF
		
		
		
	IF (stepnumber <> current_stepnumber) THEN
	
		// --- LAST SCAN ---
	
	
	END_IF
	

END_IF 

	
// Step 890
//___phase_example_Step_890_
//================================
// test dot-format from Linked EM in evaluation =>should stay in dot-format 
//================================	  

IF (stepnumber = 890) THEN

	
	IF (first_scan) THEN
	
		// --- FIRST SCAN ---
		

	ELSE
	
		// --- CONTINUOUS ---
		

	END_IF
	
	
	// --- TRANSITION TO S910 ---
	IF (
		Some_Dyn_EM.Level >= 50.0
	) THEN
	
		stepnumber:= 910;
		
	END_IF
		
		
		
	IF (stepnumber <> current_stepnumber) THEN
	
		// --- LAST SCAN ---
	
	
	END_IF
	

END_IF 

	
// Step 910
//___phase_example_Step_910_
//================================
// test suffix-format to Linked EM in assignment => should convert to dot-format
// Some_Dyn_EM_P_SP  = 4.3
// Not longer supported: only support dot notation because it is more natural to use. Keep it simple. 
//================================	  

IF (stepnumber = 910) THEN

	
	IF (first_scan) THEN
	
		// --- FIRST SCAN ---
		

	ELSE
	
		// --- CONTINUOUS ---
		

	END_IF
	
	
	// --- TRANSITION TO S920 ---
	IF (
		TRUE
	) THEN
	
		stepnumber:= 920;
		
	END_IF
		
		
		
	IF (stepnumber <> current_stepnumber) THEN
	
		// --- LAST SCAN ---
	
	
	END_IF
	

END_IF 

	
// Step 920
//___phase_example_Step_920_
//================================
// test suffix-format from Linked EM in evaluation =>should convert to dot-format
// Cancelled support for this: simplify and only allow dot format 
//================================	  

IF (stepnumber = 920) THEN

	
	IF (first_scan) THEN
	
		// --- FIRST SCAN ---
		

	ELSE
	
		// --- CONTINUOUS ---
		

	END_IF
	
	
	// --- TRANSITION TO S930 ---
	IF (
		TRUE
	) THEN
	
		stepnumber:= 930;
		
	END_IF
		
		
		
	IF (stepnumber <> current_stepnumber) THEN
	
		// --- LAST SCAN ---
	
	
	END_IF
	

END_IF 

	
// Step 930
//___phase_example_Step_930_
//================================
// write a bool 
//================================	  

IF (stepnumber = 930) THEN

	
	IF (first_scan) THEN
	
		// --- FIRST SCAN ---
		

	ELSE
	
		// --- CONTINUOUS ---
		

		// Action: some_bool_out = true
		some_bool_out:= true;

	END_IF
	
	
	// --- TRANSITION TO S940 ---
	IF (
		TRUE
	) THEN
	
		stepnumber:= 940;
		
	END_IF
		
		
		
	IF (stepnumber <> current_stepnumber) THEN
	
		// --- LAST SCAN ---
	
	
	END_IF
	

END_IF 

	
// Step 940
//___phase_example_Step_940_
//================================
// test absolute value calculation 
//================================	  

IF (stepnumber = 940) THEN

	
	IF (first_scan) THEN
	
		// --- FIRST SCAN ---
		

	ELSE
	
		// --- CONTINUOUS ---
		

		// Action: test1 = abs(2.3)
		test1:= abs(2.3);

		// Action: test2 = abs(test1)
		test2:= abs(test1);

	END_IF
	
	
	// --- TRANSITION TO S950 ---
	IF (
		TRUE
	) THEN
	
		stepnumber:= 950;
		
	END_IF
		
		
		
	IF (stepnumber <> current_stepnumber) THEN
	
		// --- LAST SCAN ---
	
	
	END_IF
	

END_IF 

	
// Step 950
//___phase_example_Step_950_
//================================
// test absolute value calculation to int value 
//================================	  

IF (stepnumber = 950) THEN

	
	IF (first_scan) THEN
	
		// --- FIRST SCAN ---
		

	ELSE
	
		// --- CONTINUOUS ---
		

		// Action: intvar = abs(4.6)
		intvar:= REAL_TO_INT( abs(4.6) );

		// Action: intvar = abs(test1)
		intvar:= REAL_TO_INT( abs(test1) );

		// Action: intvar = intvar + (intvar+ abs(3.2))
		intvar:= REAL_TO_INT( intvar + (intvar + abs(3.2)) );

	END_IF
	
	
	// --- TRANSITION TO S960 ---
	IF (
		TRUE
	) THEN
	
		stepnumber:= 960;
		
	END_IF
		
		
		
	IF (stepnumber <> current_stepnumber) THEN
	
		// --- LAST SCAN ---
	
	
	END_IF
	

END_IF 

	
// Step 960
//___phase_example_Step_960_
//================================
// test absolut function of another calc 
//================================	  

IF (stepnumber = 960) THEN

	
	IF (first_scan) THEN
	
		// --- FIRST SCAN ---
		

	ELSE
	
		// --- CONTINUOUS ---
		

		// Action: test1 = abs(test1 + test2)
		test1:= abs(test1 + test2);

	END_IF
	
	
	// --- TRANSITION TO S970 ---
	IF (
		TRUE
	) THEN
	
		stepnumber:= 970;
		
	END_IF
		
		
		
	IF (stepnumber <> current_stepnumber) THEN
	
		// --- LAST SCAN ---
	
	
	END_IF
	

END_IF 

	
// Step 970
//___phase_example_Step_970_
//================================
// test multiple transitions in one step 
//================================	  

IF (stepnumber = 970) THEN

	
	IF (first_scan) THEN
	
		// --- FIRST SCAN ---
		

	ELSE
	
		// --- CONTINUOUS ---
		

	END_IF
	
	
	// --- TRANSITION TO S980 ---
	IF (
		foo > 1.0
	) THEN
	
		stepnumber:= 980;
		
	END_IF
		
		
	// --- TRANSITION TO S990 ---
	IF (
		foo <= 1.0
	) THEN
	
		stepnumber:= 990;
		
	END_IF
		
		
		
	IF (stepnumber <> current_stepnumber) THEN
	
		// --- LAST SCAN ---
	
	
	END_IF
	

END_IF 

	
// Step 980
//___phase_example_Step_980_
//================================
// assignment where the right part is a boolean variable 
//================================	  

IF (stepnumber = 980) THEN

	
	IF (first_scan) THEN
	
		// --- FIRST SCAN ---
		

	ELSE
	
		// --- CONTINUOUS ---
		

		// Action: Bool1 = Bool2
		Bool1:= Bool2;

	END_IF
	
	
	// --- TRANSITION TO S990 ---
	IF (
		TRUE
	) THEN
	
		stepnumber:= 990;
		
	END_IF
		
		
		
	IF (stepnumber <> current_stepnumber) THEN
	
		// --- LAST SCAN ---
	
	
	END_IF
	

END_IF 

	
// Step 990
//___phase_example_Step_990_
//================================
// comparison where the right part is a boolen variable 
//================================	  

IF (stepnumber = 990) THEN

	
	IF (first_scan) THEN
	
		// --- FIRST SCAN ---
		

	ELSE
	
		// --- CONTINUOUS ---
		

	END_IF
	
	
	// --- TRANSITION TO S1000 ---
	IF (
		Bool1 = Bool2
	) THEN
	
		stepnumber:= 1000;
		
	END_IF
		
		
		
	IF (stepnumber <> current_stepnumber) THEN
	
		// --- LAST SCAN ---
	
	
	END_IF
	

END_IF 

	
// Step 1000
//___phase_example_Step_1000_
//================================
// function call 
//================================	  

IF (stepnumber = 1000) THEN

	
	IF (first_scan) THEN
	
		// --- FIRST SCAN ---
		

	ELSE
	
		// --- CONTINUOUS ---
		

		// Action: function call: write_to_DB_DW (50, 20, 123)
		write_to_DB_DW(
			DB_NO:= 50,
			Location:= 20,
			Value:= 123
		);

		// Action: function call: write_to_DB_DW (DB_NO, 20, 123)
		write_to_DB_DW(
			DB_NO:= DB_NO,
			Location:= 20,
			Value:= 123
		);

		// Action: function call: intvar = somefunction(34,32)
		intvar:= somefunction(
			arg1:= 34,
			arg2:= 32
		);

	END_IF
	
	
	// --- TRANSITION TO S0 ---
	IF (
		TRUE
	) THEN
	
		stepnumber:= 0;
		
	END_IF
		
		
		
	IF (stepnumber <> current_stepnumber) THEN
	
		// --- LAST SCAN ---
	
	
	END_IF
	

END_IF 

	




// Step 8000
//___phase_example_Step_8000_
//================================
// Holding 
//================================	  

IF (stepnumber = 8000) THEN

	
	IF (first_scan) THEN
	
		// --- FIRST SCAN ---
		

	ELSE
	
		// --- CONTINUOUS ---
		

	END_IF
	
	
	// --- TRANSITION TO S8990 ---
	IF (
		TRUE
	) THEN
	
		stepnumber:= 8990;
		
	END_IF
		
		
		
	IF (stepnumber <> current_stepnumber) THEN
	
		// --- LAST SCAN ---
	
	
	END_IF
	

END_IF 

	





// END OF THE STEPS AND TRANSITIONS
//################################
//################################
// Placeholder network to indicate the end of the actual sequence
//################################	  
//################################


// Write EMs
//--------------------------------
//
//--------------------------------

// TODO


                  
END_FUNCTION_BLOCK

PROGRAM prog

                    


// put some EM IDs in the phases for testing
cstate.Phases.phase_1.EM_I_OUT_ID:= 26;
cstate.Phases.phase_1.Some_Dyn_EM_ID:= 27;					


cstate.Phases.phase_2.EM_I_OUT_ID:= 28;
cstate.Phases.phase_2.Some_Dyn_EM_ID:= 29;						
				

cstate.Control_Modules();
cstate.Equipment_Modules();
cstate.Phases();


                  
END_PROGRAM

FUNCTION_BLOCK Control_Modules
  VAR
    XV001 : Valve;
    XV002 : Valve;
    XV003 : Valve;
    XV004 : Valve;
    XV300 : Valve;
    XV400 : Valve;
    XV500 : Valve;
    XV301 : Valve;
    XV501 : Valve;
    XV401 : Valve;
    MV001 : Valve;
    MV002 : Valve;
    MV003 : Valve;
    MV004 : Valve;
    MV005 : Valve;
    MV006 : Valve;
    MV007 : Valve;
    P100 : Motor;
    P200 : Motor;
    P101 : Motor;
    P201 : Motor;
    M100 : Motor_VFD;
    M101 : Motor_VFD;
    M102 : Motor_VFD;
    M103 : Motor_VFD;
    M104 : Motor_VFD;
    M105 : Motor_VFD;
    M106 : Motor_VFD;
    LT001 : AI;
    LT002 : AI;
    LT003 : AI;
    LT004 : AI;
    LT005 : AI;
    LT006 : AI;
    LT007 : AI;
    LT100 : AI;
    LT200 : AI;
    LT101 : AI;
    LT201 : AI;
    LS001 : DI;
    LS002 : DI;
    LIC001 : PID;
    LIC002 : PID;
    LIC003 : PID;
    LIC004 : PID;
    LIC005 : PID;
    LIC006 : PID;
    FIC100 : PID;
    FIC101 : PID;
  END_VAR

                    
XV001();
XV002();
XV003();
XV004();
XV300();
XV400();
XV500();
XV301();
XV501();
XV401();
MV001();
MV002();
MV003();
MV004();
MV005();
MV006();
MV007();
P100();
P200();
P101();
P201();
M100();
M101();
M102();
M103();
M104();
M105();
M106();
LT001();
LT002();
LT003();
LT004();
LT005();
LT006();
LT007();
LT100();
LT200();
LT101();
LT201();
LS001();
LS002();
LIC001();
LIC002();
LIC003();
LIC004();
LIC005();
LIC006();
FIC100();
FIC101();
					
                  
END_FUNCTION_BLOCK

FUNCTION_BLOCK Equipment_Modules
  VAR_INPUT
    EM_Instance_1 : EM_I_OUT;
    EM_Instance_2 : EM_I_OUT;
    EM_Instance_3 : EM_I_OUT;
    EM_Instance_4 : EM_I_OUT;
    EM_Instance_5 : EM_I_OUT;
    EM_Instance_6 : EM_I_OUT;
    EM_Instance_7 : EM_I_OUT;
    EM_Instance_8 : EM_I_OUT;
    EM_Instance_9 : EM_I_OUT;
    EM_Instance_10 : EM_I_OUT;
    EM_Instance_11 : EM_I_OUT;
    EM_Instance_12 : EM_I_OUT;
    EM_Instance_13 : EM_I_OUT;
    EM_Instance_14 : EM_I_OUT;
  END_VAR

                    
					
					
EM_Instance_1.EM_ID:= 26;
cstate.EM_Index[26]:= ADR(EM_Instance_1);
EM_Instance_1();
					
EM_Instance_2.EM_ID:= 27;
cstate.EM_Index[27]:= ADR(EM_Instance_2);
EM_Instance_2();
					
EM_Instance_3.EM_ID:= 28;
cstate.EM_Index[28]:= ADR(EM_Instance_3);
EM_Instance_3();
					
EM_Instance_4.EM_ID:= 29;
cstate.EM_Index[29]:= ADR(EM_Instance_4);
EM_Instance_4();
					
EM_Instance_5.EM_ID:= 30;
cstate.EM_Index[30]:= ADR(EM_Instance_5);
EM_Instance_5();
					
EM_Instance_6.EM_ID:= 31;
cstate.EM_Index[31]:= ADR(EM_Instance_6);
EM_Instance_6();
					
EM_Instance_7.EM_ID:= 32;
cstate.EM_Index[32]:= ADR(EM_Instance_7);
EM_Instance_7();
					
EM_Instance_8.EM_ID:= 33;
cstate.EM_Index[33]:= ADR(EM_Instance_8);
EM_Instance_8();
					
EM_Instance_9.EM_ID:= 34;
cstate.EM_Index[34]:= ADR(EM_Instance_9);
EM_Instance_9();
					
EM_Instance_10.EM_ID:= 35;
cstate.EM_Index[35]:= ADR(EM_Instance_10);
EM_Instance_10();
					
EM_Instance_11.EM_ID:= 36;
cstate.EM_Index[36]:= ADR(EM_Instance_11);
EM_Instance_11();
					
EM_Instance_12.EM_ID:= 37;
cstate.EM_Index[37]:= ADR(EM_Instance_12);
EM_Instance_12();
					
EM_Instance_13.EM_ID:= 38;
cstate.EM_Index[38]:= ADR(EM_Instance_13);
EM_Instance_13();
					
EM_Instance_14.EM_ID:= 39;
cstate.EM_Index[39]:= ADR(EM_Instance_14);
EM_Instance_14();
										

					
                  
END_FUNCTION_BLOCK

FUNCTION_BLOCK Phases
  VAR_INPUT
    phase_1 : phase_example;
    phase_2 : phase_example;
  END_VAR

                    
					
					
phase_1();
					
phase_2();
										

					
                  
END_FUNCTION_BLOCK

CONFIGURATION Application
  RESOURCE App ON PLC
    {attribute 'qualified_only'}
    VAR_GLOBAL  (* cstate *)
      Phases : Phases;
      Equipment_Modules : Equipment_Modules;
      Control_Modules : Control_Modules;
      EM_Index : ARRAY[0..300] OF DWORD;
    END_VAR
    TASK Main(INTERVAL := T#200ms, PRIORITY := 1);
    PROGRAM prog WITH Main : prog;
  END_RESOURCE
END_CONFIGURATION
